# B&R Automation Studio project ABC_Pltzr
Automation Studio 3.0.90.24 SP06


## Configuration PPC70_JOB24025

CPU 4PPC70.101G-20F005, AutomationRuntime D4.22, Build 4.1.2, Vc V4.24.0, Safety 0.0

### Hardware
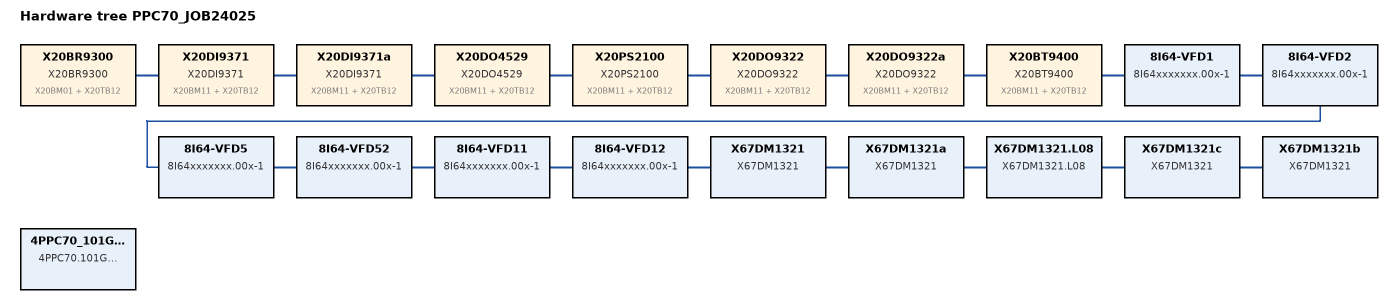
```
4PPC70_101G_20F005 : 4PPC70.101G-20F005 v1.1.0.0
  Connector IF1:
    ActivatePowerlink = 0
  Connector IF2:
    ActivateDevice = 1
    Mode = Manual
    InternetAddress = 192.168.1.100
    SubnetMask = 255.255.255.0
    InaNodeNumber = 1
    Vnc1
    VncVcObjectName1 = WSVGA
    VncKeyMappingFile1 = VC\PS2-Keyboard.dis
    VncAuthentication1 = 1
    VncPasswordViewOnly1 = v
    VncPasswordViewControl1 = 24025
    VncMaxConnections1 = 2
    VncRefreshRate1 = 500
  PermanentPvSize = 1000
  RemanentGlobalPvSize = 25000
  VolatileGlobalPvSize = 200000
  EnableUsbRemoteInstall = 1
  TimerDeviceType = SWIOTIMER
  Cyclic1Duration = 4000
  Cyclic1Tolerance = 4000
  Cyclic2Duration = 20000
  Cyclic2Tolerance = 20000
  Cyclic3Duration = 50000
  Cyclic3Tolerance = 50000
  Cyclic4Duration = 100000
  Cyclic4Tolerance = 100000
  Cyclic5Duration = 200000
  Cyclic5Tolerance = 200000
  Cyclic6Duration = 500000
  Cyclic6Tolerance = 500000
  Cyclic7Duration = 1000000
  Cyclic7Tolerance = 1000000
  Cyclic8Duration = 10000
  Cyclic8Tolerance = 30000000
  FtpUser1
  FtpUsername1 = abc
  FtpUserPassword1 = veVz20Da1KUF2Vww53L6omFNdzfk8lHY0HjcrjfOb/w=  // abc123
  FtpUserSalt1 = pyAcjG26
  FTPPath1 = 5
  FTPAccessRight1 = 0
  VcObjectName = WSVGA
  KeyMappingFile = VC\4PPC70_101G_20F005.dis
8I64-VFD1 : 8I64xxxxxxx.00x-1 v1.3.8.1  [X2X1 -> X20BT9400.X2X1]
  FunctionModel = Standard
  Supervision = off
  enableIOLR = off
  enableDigitalOutput = off
  DigitalOutputMode01 = actionDO
  ACC = 1
  DEC = 1
  HSP = 900
  ITH = 28
  BFR = 1
  UNS = 460
  FRS = 600
  NCR = 28
  NSP = 1750
  COS = 80
  TFR = 900
  DO = 9
  BRA = 0
  BLC = 64
  BRT = 15
  BEN = 0
  BET = 15
8I64-VFD11 : 8I64xxxxxxx.00x-1 v1.3.8.1  [X2X1 -> 8I64-VFD52.X2X2]
  FunctionModel = Standard
  Supervision = off
  enableIOLR = off
  enableDigitalOutput = off
  DigitalOutputMode01 = actionDO
  DownloadParameters = yes
  ACC = 1
  DEC = 1
  HSP = 900
  ITH = 13
  FTD = 600
  BFR = 1
  UNS = 460
  FRS = 600
  NCR = 13
  NSP = 1750
  COS = 80
  TFR = 900
  DO = 9
  BRA = 0
  BLC = 64
  BRT = 5
  BEN = 0
  BET = 5
8I64-VFD12 : 8I64xxxxxxx.00x-1 v1.3.8.1  [X2X1 -> 8I64-VFD11.X2X2]
  FunctionModel = Standard
  Supervision = off
  enableIOLR = off
  enableDigitalOutput = off
  DigitalOutputMode01 = actionDO
  DownloadParameters = yes
  ACC = 1
  DEC = 200
  HSP = 900
  ITH = 13
  FTD = 600
  BFR = 1
  UNS = 460
  FRS = 600
  NCR = 13
  NSP = 1750
  COS = 80
  TFR = 900
  DO = 9
  BRA = 0
  BLC = 64
  BRT = 5
  BEN = 0
  BET = 5
8I64-VFD2 : 8I64xxxxxxx.00x-1 v1.3.8.1  [X2X1 -> 8I64-VFD1.X2X2]
  FunctionModel = Standard
  Supervision = off
  enableIOLR = off
  enableDigitalOutput = off
  DigitalOutputMode01 = actionDO
  DownloadParameters = yes
  ACC = 1
  DEC = 1
  HSP = 900
  BFR = 1
  UNS = 460
  FRS = 600
  NCR = 13
  NSP = 1750
  TFR = 900
  DO = 9
  BRA = 0
  BLC = 64
  BRT = 5
  BEN = 0
  BET = 5
8I64-VFD5 : 8I64xxxxxxx.00x-1 v1.3.8.1  [X2X1 -> 8I64-VFD2.X2X2]
  FunctionModel = Standard
  Supervision = off
  DownloadParameters = yes
  ACC = 1
  DEC = 1
  HSP = 900
  ITH = 13
  FTD = 600
  BFR = 1
  UNS = 460
  FRS = 600
  NCR = 13
  NSP = 1750
  COS = 80
  TFR = 900
  DE2 = 10
  BRA = 0
8I64-VFD52 : 8I64xxxxxxx.00x-1 v1.3.8.1  [X2X1 -> 8I64-VFD5.X2X2]
  FunctionModel = Standard
  Supervision = off
  enableIOLR = off
  enableDigitalOutput = off
  DigitalOutputMode01 = actionDO
  ACC = 1
  DEC = 1
  HSP = 900
  ITH = 13
  FTD = 600
  BFR = 1
  UNS = 460
  FRS = 600
  NCR = 13
  NSP = 1750
  COS = 80
  TFR = 900
  DO = 9
  INR = 0
  BRA = 0
  BLC = 64
  BRT = 1
  BEN = 0
  BET = 1
X20BM01 : X20BM01 v1.0.0.1
X20BM11 : X20BM11 v1.0.0.0  [X2X1 -> X20BM01.X2X2]
X20BM11a : X20BM11 v1.0.0.0  [X2X1 -> X20BM11.X2X2]
X20BM11b : X20BM11 v1.0.0.0  [X2X1 -> X20BM11a.X2X2]
X20BM11c : X20BM11 v1.0.0.0  [X2X1 -> X20BM11b.X2X2]
X20BM11d : X20BM11 v1.0.0.0  [X2X1 -> X20BM11c.X2X2]
X20BM11e : X20BM11 v1.0.0.0  [X2X1 -> X20BM11f.X2X2]
X20BM11f : X20BM11 v1.0.0.0  [X2X1 -> X20BM11d.X2X2]
X20BR9300 : X20BR9300 v1.0.2.6  [SS1 -> X20TB12.SS; SL -> X20BM01.SL1; X2X1 -> 4PPC70_101G_20F005.IF5]
  Supervision = off
X20BT9400 : X20BT9400 v1.0.1.3  [SS1 -> X20TB12f.SS; SL -> X20BM11e.SL1]
  Supervision = off
X20DI9371 : X20DI9371 v1.0.1.2  [SS1 -> X20TB12a.SS; SL -> X20BM11.SL1]
  Supervision = off
X20DI9371a : X20DI9371 v1.0.1.2  [SS1 -> X20TB12b.SS; SL -> X20BM11a.SL1]
  Supervision = off
  InputFilter = 100
X20DO4529 : X20DO4529 v1.0.1.2  [SS1 -> X20TB12c.SS; SL -> X20BM11b.SL1]
  Supervision = off
X20DO9322 : X20DO9322 v1.0.2.2  [SS1 -> X20TB12e.SS; SL -> X20BM11d.SL1]
  Supervision = off
X20DO9322a : X20DO9322 v1.0.2.2  [SS1 -> X20TB12g.SS; SL -> X20BM11f.SL1]
  Supervision = off
X20PS2100 : X20PS2100 v1.0.3.0  [SS1 -> X20TB12d.SS; SL -> X20BM11c.SL1]
  Supervision = off
X20TB12 : X20TB12 v1.0.0.0
X20TB12a : X20TB12 v1.0.0.0
X20TB12b : X20TB12 v1.0.0.0
X20TB12c : X20TB12 v1.0.0.0
X20TB12d : X20TB12 v1.0.0.0
X20TB12e : X20TB12 v1.0.0.0
X20TB12f : X20TB12 v1.0.0.0
X20TB12g : X20TB12 v1.0.0.0
X67DM1321 : X67DM1321 v1.1.1.0  [X2X1 -> 8I64-VFD12.X2X2]
  Supervision = off
X67DM1321.L08 : X67DM1321.L08 v1.1.2.0  [X2X1 -> X67DM1321a.X2X2]
  Supervision = off
  Direction01 = output
  Direction02 = output
  Direction03 = output
  Direction04 = output
  Direction05 = output
  Direction06 = output
  Direction07 = output
  Direction08 = output
  Direction09 = output
  Direction10 = output
  Direction11 = output
  Direction12 = output
X67DM1321a : X67DM1321 v1.1.1.0  [X2X1 -> X67DM1321.X2X2]
  Supervision = off
  Direction01 = output
  Direction02 = output
  Direction03 = output
  Direction04 = output
X67DM1321b : X67DM1321 v1.1.1.0  [X2X1 -> X67DM1321c.X2X2]
  Supervision = off
X67DM1321c : X67DM1321 v1.1.1.0  [X2X1 -> X67DM1321.L08.X2X2]
  Supervision = off
  Direction01 = output
  Direction02 = output
```


## Logical view

Binary libraries used (declarations not repeated): astime, DataObj, Ethernet, MpCom 1.20.3, sys_lib, CSV_File

### appConfigAndRecipes.var
```iecst
(********************************************************************
 * COPYRIGHT --
 ********************************************************************
 * Package: ConfigAndRecipes
 * File: ConfigAndRecipes.var
 * Author: goran_2
 * Created: August 06, 2011
 ********************************************************************
 * Variables of package ConfigAndRecipes
 ********************************************************************)
VAR RETAIN
	gRecipe : paiRecipeApp_typ := (0);
END_VAR
VAR
	gPVSerDesMgr : paiPVSerDesMgr_typ := (0);
	gSerDesHMI_gConfigApp : paiPVSerDesHMI_typ := (0);
	gSerDesHMI_gPalletCfg : paiPVSerDesHMI_typ := (0);
	gSerDesMem_gConfigApp : configApp_typ := (0);
	gSerDesMem_gLayerEditor : palleteCfgLayer_typ := (0);
	gSerDesMem_gPallete_palCfg : palleteCfg_typ := (0);
	gDummy : UDINT := 0;
END_VAR
```

### appCfgRecDefault.h
```c
/********************************************************************
 * COPYRIGHT -- HP
 ********************************************************************
 * Program: cfgFS
 * File: cfgFSApp.h
 * Author: goran
 * Created: March 19, 2014
 *******************************************************************/

#include <bur/plctypes.h>

/*
###############################################################################
Defines, Consts
###############################################################################
*/
/*
NOTE: Using C: disk is not the best solution considering that system files are there.
However, using disk other then C: (i.e. D:, etc) for application stuff creates
issue with the ability to view/copy/access application files from windows (multiple partitions not supported, etc)

File structure used in this application is following:

Directory:
C://Data
is used for application specific stuff.
This directory holds following files:
machine configuration file - "appcfg.txt"
machine factory deafult configuration file - "appcfgfactory.txt");

a subdirectory (REC) of the above directory is used for storing recipes.
C://Data/Rec

*/

#define APP_FILE_SIZE_MAX  30000 //max file size for any recipe or config file

#define APP_DIR_NAME "Data" //root app directory; Example: C://Data
#define APP_REC_DIR_NAME "Rec" // recipes directory; Example "C://Data/Rec"

#define APP_FILENAME_CFG "appcfg.txt"
#define APP_FILENAME_CFGDEFAULT "appcfgfactory.txt"
#define APP_FILENAME_CURRECIPE "apprec.txt"
```

### Alarms.typ
```iecst
(********************************************************************

 * COPYRIGHT -- Piedmont Automation Inc.

 ********************************************************************

 * File: Alarms.typ

 * Author: goran

 * Created: Jun 1, 2015

 ********************************************************************

 * Data types for project : Alarms

 ********************************************************************)

TYPE
	applicationAlarms_enums :
		(
		APP_ALARM_HWMODULE := 0,
		APP_ALARM_DS1,
		APP_ALARM_DS2,
		APP_ALARM_DS3,
		APP_ALARM_DS4,
		APP_ALARM_DS5,
		APP_ALARM_DS6,
		APP_ALARM_ESTOP1,
		APP_ALARM_ESTOP2,
		APP_ALARM_ESTOP3,
		APP_ALARM_ESTOP4,
		APP_ALARM_ESTOP5,
		APP_ALARM_ESTOP6,
		APP_ALARM_MOTOROL,
		APP_ALARM_MCR,
		APP_ALARM_AIRPRESSURE,
		APP_ALARM_ELEV_CHAINSLACK_LF,
		APP_ALARM_ELEV_CHAINSLACK_RT,
		APP_ALARM_ELEV_PALLETDISPENS,
		APP_ALARM_VFD,
		APP_ALARM_LIGHT_CURTAIN_OSSD1,
		APP_ALARM_LIGHT_CURTAIN_OSSD2,
		APP_ALARM_INFEED_JAM,
		APP_ALARM_ROW_FORMING_JAM,
		APP_ALARM_ROW_TOO_LONG,
		APP_ALARM_INVALID_PROGRAM,
		APP_ALARM_PALLET_EXIT_TIMEOUT,
		APP_ALARM_INFEED_CASE_COUNT,
		APP_ALARM_LASTTOCHECK := 48,
		APP_ALARM_ALARMACKNEEDED := 49,
		APP_ALARM_LAST := 50
		);
END_TYPE

(*########################################################################*)
(*Application object - Alarm Object*)
(*########################################################################*)

TYPE
	applicationAlarms_typ : 	STRUCT
		oIsAlarmActiveCount : UDINT; (*1-if alarm present*)
		oIsAlarmNotAckCount : UDINT; (*1-if not ack alarm present*)
		oIsAlarmActive : BOOL; (*1-if alarm present*)
		oIsAlarmNotAck : BOOL; (*1-if not ack alarm present*)
		alarmActive : ARRAY[0..APP_ALARM_LAST]OF BOOL; (*Alarms matrix. (see Visual Components Alarm System)*)
		alarmAck : ARRAY[0..APP_ALARM_LAST]OF BOOL; (*Alarms ack matrix. (see Visual Components Alarm System)*)
	END_STRUCT;
END_TYPE
```

- appOffOnColor.clm (not shown)

- lightFeature.clm (not shown)

- pageTabs.clm (not shown)

- paiPingStatus.clm (not shown)

- Arial12px.fninfo (not shown)

- Arial7px.fninfo (not shown)

- Status_0.fninfo (not shown)

- paiHmiMenu.layer (not shown)

### sscanf2.h
```c
/********************************************************
*	NAME	: sscanf2.h
*	FUNCTION: Headerfile for the sscanf2.a implementation
*			  of the standard "C" function: sscanf().
*********************************************************/

extern int sscanf2(char *s, char *fmt, ...);
```

### Program Logical/MachineControl/blades

#### Cyclic.ld
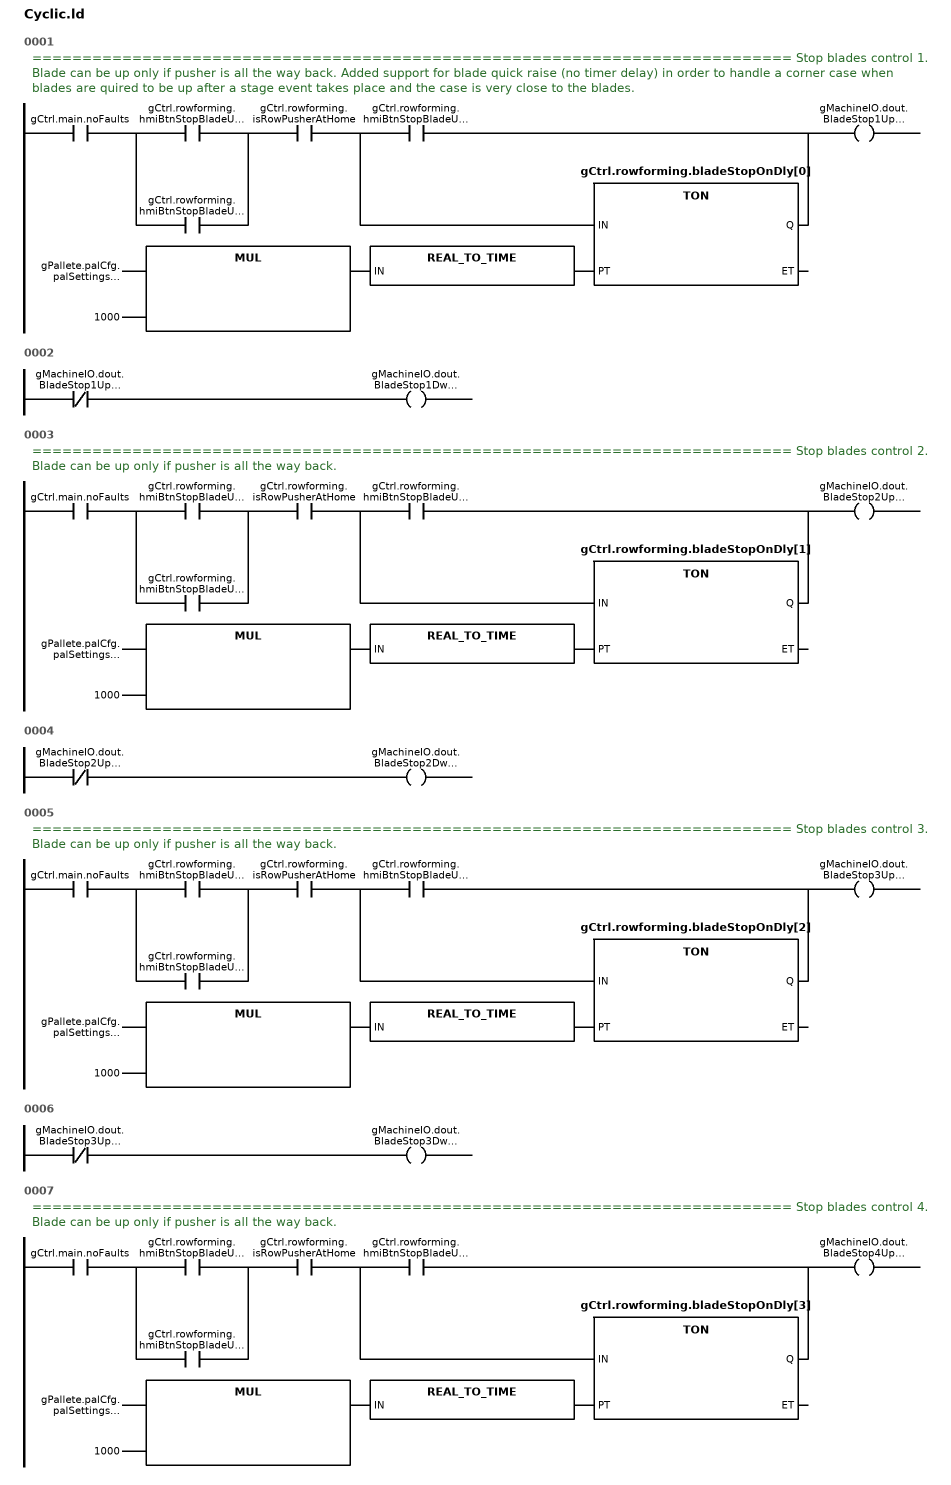
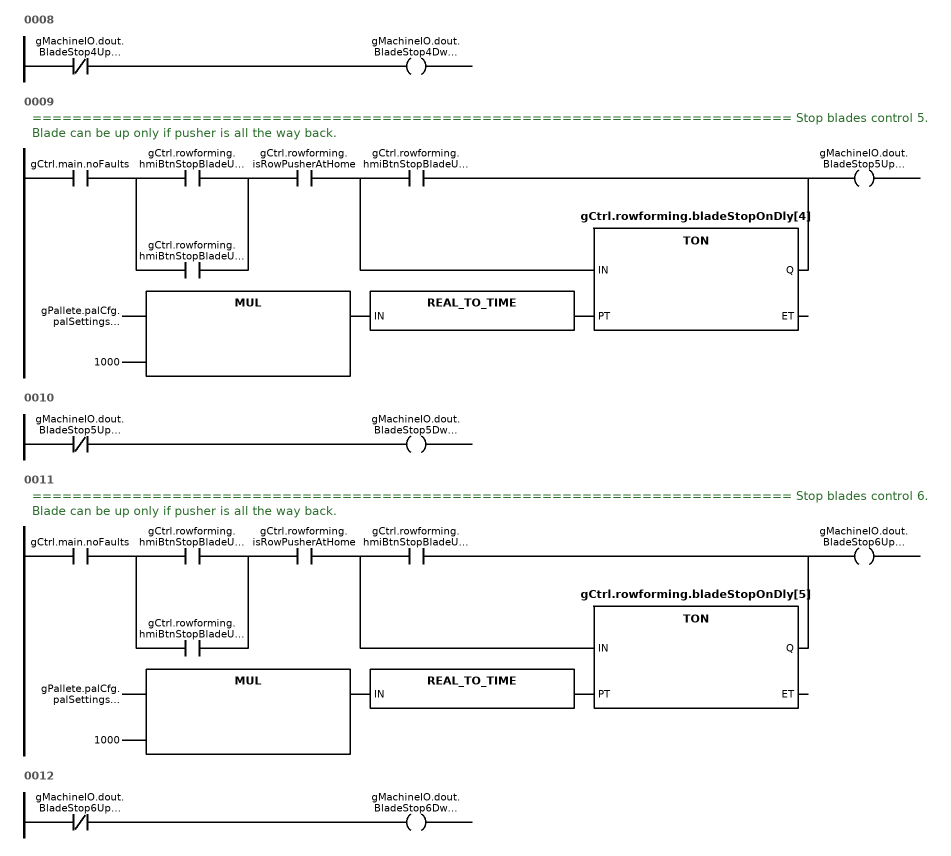
Ladder, written as Structured Text:
```iecst
PROGRAM _CYCLIC
VAR
    _p1 : BOOL;
    _p2 : BOOL;
    _p3 : BOOL;
    _p4 : BOOL;
    _p5 : BOOL;
    _p6 : BOOL;
END_VAR
(* Network 1: ============================================================================ Stop blades control 1. Blade can be up only if pusher is all the way back. Added support for blade quick raise (no timer delay) in order to handle a corner case when blades are quired to be up after a stage event takes place and the case is very close to the blades. *)
_p1 := gCtrl.main.noFaults AND (gCtrl.rowforming.hmiBtnStopBladeUpDown1 OR gCtrl.rowforming.hmiBtnStopBladeUpDownQuick1) AND gCtrl.rowforming.isRowPusherAtHome;
gMachineIO.dout.BladeStop1Up_SOL3A := (_p1 AND gCtrl.rowforming.hmiBtnStopBladeUpDownQuick1) OR gCtrl.rowforming.bladeStopOnDly[0].Q;
gCtrl.rowforming.bladeStopOnDly[0](IN := _p1, PT := REAL_TO_TIME(gPallete.palCfg.palSettings.timers.bladeStopOnDly1 * 1000));

(* Network 2 *)
gMachineIO.dout.BladeStop1Dw_SOL3B := NOT gMachineIO.dout.BladeStop1Up_SOL3A;

(* Network 3: ============================================================================ Stop blades control 2. Blade can be up only if pusher is all the way back. *)
_p2 := gCtrl.main.noFaults AND (gCtrl.rowforming.hmiBtnStopBladeUpDown2 OR gCtrl.rowforming.hmiBtnStopBladeUpDownQuick2) AND gCtrl.rowforming.isRowPusherAtHome;
gMachineIO.dout.BladeStop2Up_SOL4A := (_p2 AND gCtrl.rowforming.hmiBtnStopBladeUpDownQuick2) OR gCtrl.rowforming.bladeStopOnDly[1].Q;
gCtrl.rowforming.bladeStopOnDly[1](IN := _p2, PT := REAL_TO_TIME(gPallete.palCfg.palSettings.timers.bladeStopOnDly2 * 1000));

(* Network 4 *)
gMachineIO.dout.BladeStop2Dw_SOL4B := NOT gMachineIO.dout.BladeStop2Up_SOL4A;

(* Network 5: ============================================================================ Stop blades control 3. Blade can be up only if pusher is all the way back. *)
_p3 := gCtrl.main.noFaults AND (gCtrl.rowforming.hmiBtnStopBladeUpDown3 OR gCtrl.rowforming.hmiBtnStopBladeUpDownQuick3) AND gCtrl.rowforming.isRowPusherAtHome;
gMachineIO.dout.BladeStop3Up_SOL5A := (_p3 AND gCtrl.rowforming.hmiBtnStopBladeUpDownQuick3) OR gCtrl.rowforming.bladeStopOnDly[2].Q;
gCtrl.rowforming.bladeStopOnDly[2](IN := _p3, PT := REAL_TO_TIME(gPallete.palCfg.palSettings.timers.bladeStopOnDly3 * 1000));

(* Network 6 *)
gMachineIO.dout.BladeStop3Dw_SOL5B := NOT gMachineIO.dout.BladeStop3Up_SOL5A;

(* Network 7: ============================================================================ Stop blades control 4. Blade can be up only if pusher is all the way back. *)
_p4 := gCtrl.main.noFaults AND (gCtrl.rowforming.hmiBtnStopBladeUpDown4 OR gCtrl.rowforming.hmiBtnStopBladeUpDownQuick4) AND gCtrl.rowforming.isRowPusherAtHome;
gMachineIO.dout.BladeStop4Up_SOL6A := (_p4 AND gCtrl.rowforming.hmiBtnStopBladeUpDownQuick4) OR gCtrl.rowforming.bladeStopOnDly[3].Q;
gCtrl.rowforming.bladeStopOnDly[3](IN := _p4, PT := REAL_TO_TIME(gPallete.palCfg.palSettings.timers.bladeStopOnDly4 * 1000));

(* Network 8 *)
gMachineIO.dout.BladeStop4Dw_SOL6B := NOT gMachineIO.dout.BladeStop4Up_SOL6A;

(* Network 9: ============================================================================ Stop blades control 5. Blade can be up only if pusher is all the way back. *)
_p5 := gCtrl.main.noFaults AND (gCtrl.rowforming.hmiBtnStopBladeUpDown5 OR gCtrl.rowforming.hmiBtnStopBladeUpDownQuick5) AND gCtrl.rowforming.isRowPusherAtHome;
gMachineIO.dout.BladeStop5Up_SOL13A := (_p5 AND gCtrl.rowforming.hmiBtnStopBladeUpDownQuick5) OR gCtrl.rowforming.bladeStopOnDly[4].Q;
gCtrl.rowforming.bladeStopOnDly[4](IN := _p5, PT := REAL_TO_TIME(gPallete.palCfg.palSettings.timers.bladeStopOnDly5 * 1000));

(* Network 10 *)
gMachineIO.dout.BladeStop5Dw_SOL13B := NOT gMachineIO.dout.BladeStop5Up_SOL13A;

(* Network 11: ============================================================================ Stop blades control 6. Blade can be up only if pusher is all the way back. *)
_p6 := gCtrl.main.noFaults AND (gCtrl.rowforming.hmiBtnStopBladeUpDown6 OR gCtrl.rowforming.hmiBtnStopBladeUpDownQuick6) AND gCtrl.rowforming.isRowPusherAtHome;
gMachineIO.dout.BladeStop6Up_SOL14A := (_p6 AND gCtrl.rowforming.hmiBtnStopBladeUpDownQuick6) OR gCtrl.rowforming.bladeStopOnDly[5].Q;
gCtrl.rowforming.bladeStopOnDly[5](IN := _p6, PT := REAL_TO_TIME(gPallete.palCfg.palSettings.timers.bladeStopOnDly6 * 1000));

(* Network 12 *)
gMachineIO.dout.BladeStop6Dw_SOL14B := NOT gMachineIO.dout.BladeStop6Up_SOL14A;
END_PROGRAM
```

### Program Logical/MachineControl/elevator

#### Cyclic.ld
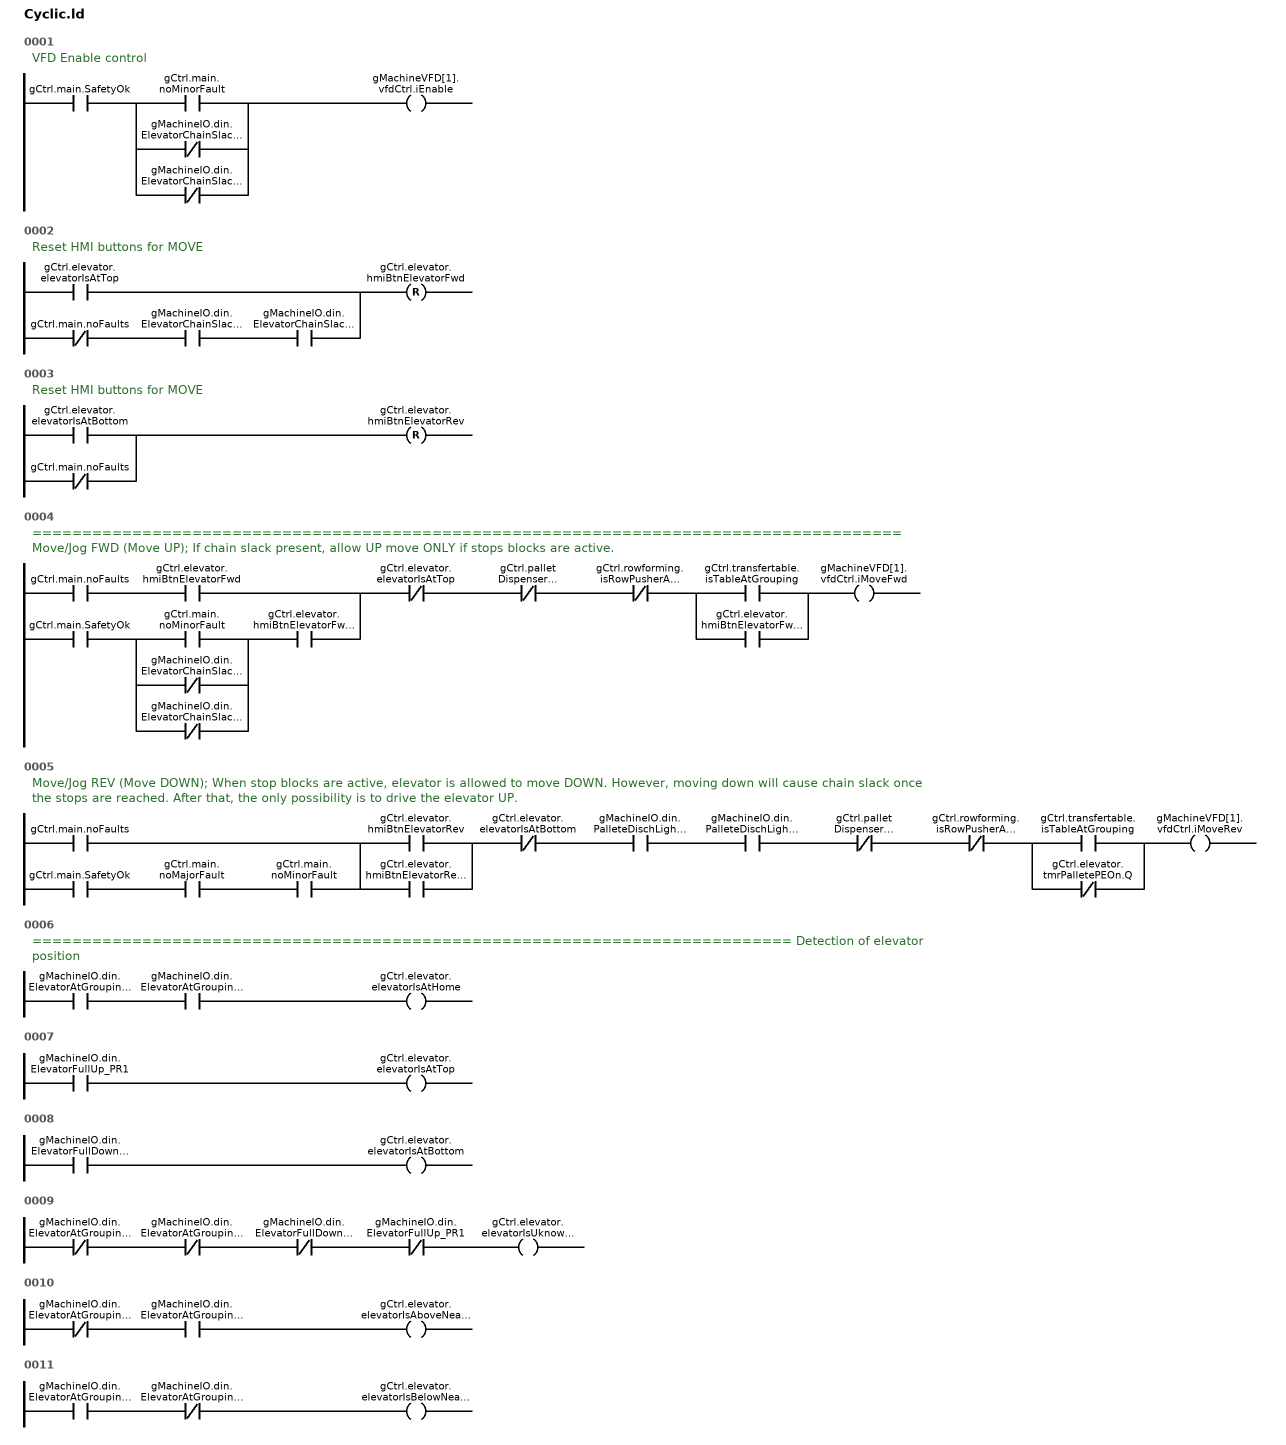
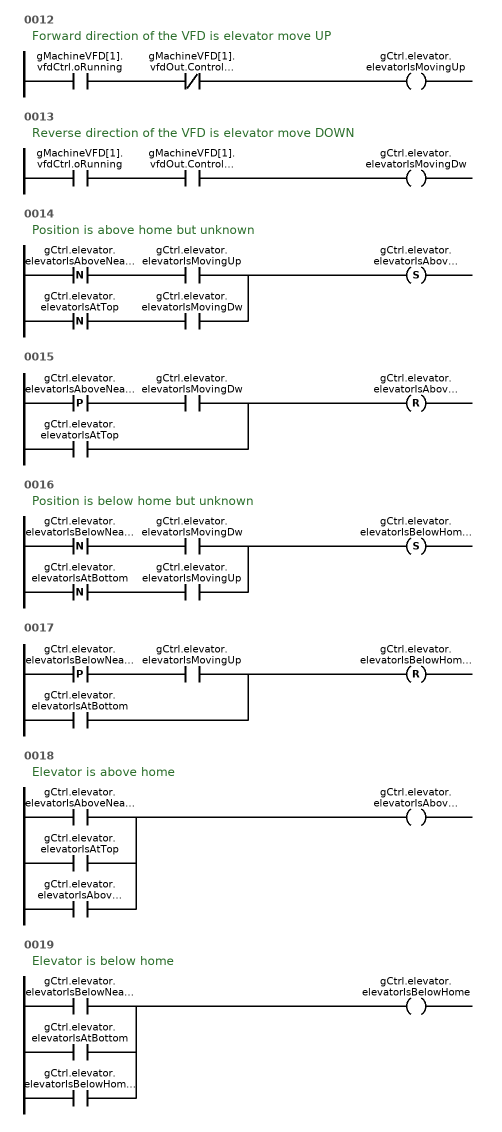
Ladder, written as Structured Text:
```iecst
PROGRAM _CYCLIC
VAR
    _p1 : BOOL;
    _p2 : BOOL;
    _p3 : BOOL;
    _e4 : F_TRIG;
    _e5 : F_TRIG;
    _e6 : R_TRIG;
    _e7 : F_TRIG;
    _e8 : F_TRIG;
    _e9 : R_TRIG;
END_VAR
(* Network 1: VFD Enable control *)
gMachineVFD[1].vfdCtrl.iEnable := gCtrl.main.SafetyOk AND (gCtrl.main.noMinorFault OR NOT gMachineIO.din.ElevatorChainSlackLF_LS7 OR NOT gMachineIO.din.ElevatorChainSlackRT_LS8);

(* Network 2: Reset HMI buttons for MOVE *)
IF gCtrl.elevator.elevatorIsAtTop OR (NOT gCtrl.main.noFaults AND gMachineIO.din.ElevatorChainSlackLF_LS7 AND gMachineIO.din.ElevatorChainSlackRT_LS8) THEN
    gCtrl.elevator.hmiBtnElevatorFwd := FALSE;
END_IF;

(* Network 3: Reset HMI buttons for MOVE *)
IF gCtrl.elevator.elevatorIsAtBottom OR NOT gCtrl.main.noFaults THEN
    gCtrl.elevator.hmiBtnElevatorRev := FALSE;
END_IF;

(* Network 4: ======================================================================================= Move/Jog FWD (Move UP); If chain slack present, allow UP move ONLY if stops blocks are active. *)
_p1 := ((gCtrl.main.noFaults AND gCtrl.elevator.hmiBtnElevatorFwd) OR (gCtrl.main.SafetyOk AND (gCtrl.main.noMinorFault OR NOT gMachineIO.din.ElevatorChainSlackLF_LS7 OR NOT gMachineIO.din.ElevatorChainSlackRT_LS8) AND gCtrl.elevator.hmiBtnElevatorFwdJog)) AND NOT gCtrl.elevator.elevatorIsAtTop AND NOT gCtrl.palletDispenser.hmiBtnPalletInCVFwd AND NOT gCtrl.rowforming.isRowPusherAtElevator;
gMachineVFD[1].vfdCtrl.iMoveFwd := _p1 AND (gCtrl.transfertable.isTableAtGrouping OR gCtrl.elevator.hmiBtnElevatorFwdJog);

(* Network 5: Move/Jog REV (Move DOWN); When stop blocks are active, elevator is allowed to move DOWN. However, moving down will cause chain slack once the stops are reached. After that, the only possibility is to drive the elevator UP. *)
_p2 := gCtrl.main.SafetyOk AND gCtrl.main.noMajorFault AND gCtrl.main.noMinorFault;
_p3 := (gCtrl.main.noFaults OR _p2) AND (gCtrl.elevator.hmiBtnElevatorRev OR gCtrl.elevator.hmiBtnElevatorRevJog) AND NOT gCtrl.elevator.elevatorIsAtBottom AND gMachineIO.din.PalleteDischLightCurtain_OSSD1 AND gMachineIO.din.PalleteDischLightCurtain_OSSD2 AND NOT gCtrl.palletDispenser.hmiBtnPalletInCVFwd AND NOT gCtrl.rowforming.isRowPusherAtElevator;
gMachineVFD[1].vfdCtrl.iMoveRev := _p3 AND (gCtrl.transfertable.isTableAtGrouping OR NOT gCtrl.elevator.tmrPalletePEOn.Q);

(* Network 6: ============================================================================ Detection of elevator position *)
gCtrl.elevator.elevatorIsAtHome := gMachineIO.din.ElevatorAtGroupingLower_PR3 AND gMachineIO.din.ElevatorAtGroupingRaise_PR4;

(* Network 7 *)
gCtrl.elevator.elevatorIsAtTop := gMachineIO.din.ElevatorFullUp_PR1;

(* Network 8 *)
gCtrl.elevator.elevatorIsAtBottom := gMachineIO.din.ElevatorFullDown_PR2;

(* Network 9 *)
gCtrl.elevator.elevatorIsUknownPosition := NOT gMachineIO.din.ElevatorAtGroupingLower_PR3 AND NOT gMachineIO.din.ElevatorAtGroupingRaise_PR4 AND NOT gMachineIO.din.ElevatorFullDown_PR2 AND NOT gMachineIO.din.ElevatorFullUp_PR1;

(* Network 10 *)
gCtrl.elevator.elevatorIsAboveNearHome := NOT gMachineIO.din.ElevatorAtGroupingLower_PR3 AND gMachineIO.din.ElevatorAtGroupingRaise_PR4;

(* Network 11 *)
gCtrl.elevator.elevatorIsBelowNearHome := gMachineIO.din.ElevatorAtGroupingLower_PR3 AND NOT gMachineIO.din.ElevatorAtGroupingRaise_PR4;

(* Network 12: Forward direction of the VFD is elevator move UP *)
gCtrl.elevator.elevatorIsMovingUp := gMachineVFD[1].vfdCtrl.oRunning AND NOT gMachineVFD[1].vfdOut.Control.Direction;

(* Network 13: Reverse direction of the VFD is elevator move DOWN *)
gCtrl.elevator.elevatorIsMovingDw := gMachineVFD[1].vfdCtrl.oRunning AND gMachineVFD[1].vfdOut.Control.Direction;

(* Network 14: Position is above home but unknown *)
_e4(CLK := gCtrl.elevator.elevatorIsAboveNearHome);
_e5(CLK := gCtrl.elevator.elevatorIsAtTop);
IF (_e4.Q AND gCtrl.elevator.elevatorIsMovingUp) OR (_e5.Q AND gCtrl.elevator.elevatorIsMovingDw) THEN
    gCtrl.elevator.elevatorIsAboveHomeUnknown := TRUE;
END_IF;

(* Network 15 *)
_e6(CLK := gCtrl.elevator.elevatorIsAboveNearHome);
IF (_e6.Q AND gCtrl.elevator.elevatorIsMovingDw) OR gCtrl.elevator.elevatorIsAtTop THEN
    gCtrl.elevator.elevatorIsAboveHomeUnknown := FALSE;
END_IF;

(* Network 16: Position is below home but unknown *)
_e7(CLK := gCtrl.elevator.elevatorIsBelowNearHome);
_e8(CLK := gCtrl.elevator.elevatorIsAtBottom);
IF (_e7.Q AND gCtrl.elevator.elevatorIsMovingDw) OR (_e8.Q AND gCtrl.elevator.elevatorIsMovingUp) THEN
    gCtrl.elevator.elevatorIsBelowHomeUnknown := TRUE;
END_IF;

(* Network 17 *)
_e9(CLK := gCtrl.elevator.elevatorIsBelowNearHome);
IF (_e9.Q AND gCtrl.elevator.elevatorIsMovingUp) OR gCtrl.elevator.elevatorIsAtBottom THEN
    gCtrl.elevator.elevatorIsBelowHomeUnknown := FALSE;
END_IF;

(* Network 18: Elevator is above home *)
gCtrl.elevator.elevatorIsAboveHome := gCtrl.elevator.elevatorIsAboveNearHome OR gCtrl.elevator.elevatorIsAtTop OR gCtrl.elevator.elevatorIsAboveHomeUnknown;

(* Network 19: Elevator is below home *)
gCtrl.elevator.elevatorIsBelowHome := gCtrl.elevator.elevatorIsBelowNearHome OR gCtrl.elevator.elevatorIsAtBottom OR gCtrl.elevator.elevatorIsBelowHomeUnknown;
END_PROGRAM
```

### Program Logical/MachineControl/vfdControl

#### vfdControl.c
```c
#include <bur/plctypes.h>

#ifdef _DEFAULT_INCLUDES
	#include <AsDefault.h>
#endif

/*
16#0000	nOF: No fault code saved
16#1000	CrF: Capacitor pre-charge detected fault or
16#1000	OLF: Motor overload or
16#1000	SOF: Motor overspeed
16#2310	OCF: Overcurrent
16#2320	OCF: Impeding short-circuit or
16#2320	OCF: Power module, specific to 15kW drives
16#2330	SCF: Motor short-circuit (to ground)
16#2340	OCF: Motor short-circuit (phase to phase)
16#3110	OSF: Line supply overvoltage
16#3120	USF: Line supply undervoltage
16#3130	PHF: Line supply phase loss
16#3310	ObF: DC bus overvoltage or
16#3310	OPF: Motor phase loss or
16#3310	OPF: Motor phase loss - 3 phases
16#4210	OHF: Drive overheating
16#5520	EEF: EEPROM memory
16#6100	InF: Internal
16#6300	CFF: Incorrect configuration (parameters) or
16#6300	CFI: Invalid configuration (parameters)
16#7300	LFF: 4 - 20 mA loss
16#7510	SLF: Modbus communication interruption
16#8100	COF: Communication interruption, line 2 (CANopen)
16#9000	EPF: External fault
16#FF00	tnF: Auto-tuning was unsuccessful
16#FF01	bLF: Brake control
16#7520	ILF: Optional internal link
16#7510	CNF: Communication interruption on the communication card
*/
static void paiVFDGetFaultText(UINT faultCode, char* pDest, UDINT destSize)
{

	switch(faultCode){
		case 0x0:
			brsstrcpy((UDINT)pDest, (UDINT)"nOF: No fault code saved");
			break;
		case 0x1000:
			brsstrcpy((UDINT)pDest, (UDINT)"CrF or OLF or SOF");
			break;
		case 0x2310:
			brsstrcpy((UDINT)pDest, (UDINT)"OCF: Overcurrent");
			break;
		case 0x2320:
			brsstrcpy((UDINT)pDest, (UDINT)"OCF: Impeding short-circuit");
			break;
		case 0x2330:
			brsstrcpy((UDINT)pDest, (UDINT)"SCF: Motor short-circuit (to ground)");
			break;
		case 0x2340:
			brsstrcpy((UDINT)pDest, (UDINT)"OCF: Motor short-circuit (phase to phase)");
			break;
		case 0x3110:
			brsstrcpy((UDINT)pDest, (UDINT)"OSF: Line supply overvoltage");
			break;
		case 0x3120:
			brsstrcpy((UDINT)pDest, (UDINT)"USF: Line supply undervoltage");
			break;
		case 0x3130:
			brsstrcpy((UDINT)pDest, (UDINT)"PHF: Line supply phase loss");
			break;
		case 0x3310:
			brsstrcpy((UDINT)pDest, (UDINT)"ObF: DC bus overvoltage or OPF");
			break;
		case 0x4210:
			brsstrcpy((UDINT)pDest, (UDINT)"OHF: Drive overheating");
			break;
		case 0x5520:
			brsstrcpy((UDINT)pDest, (UDINT)"EEF: EEPROM memory");
			break;
		case 0x6100:
			brsstrcpy((UDINT)pDest, (UDINT)"InF: Internal");
			break;
		case 0x6300:
			brsstrcpy((UDINT)pDest, (UDINT)"CFF: Incorrect configuration or CFI");
			break;
		case 0x7300:
			brsstrcpy((UDINT)pDest, (UDINT)"LFF: 4 - 20 mA loss");
			break;
		case 0x7510:
			brsstrcpy((UDINT)pDest, (UDINT)"SLF: Modbus communication interruption");
			break;
		case 0x8100:
			brsstrcpy((UDINT)pDest, (UDINT)"COF: Communication interruption, line 2 (CANopen)");
			break;
		case 0x9000:
			brsstrcpy((UDINT)pDest, (UDINT)"EPF: External fault");
			break;
		case 0xFF00:
			brsstrcpy((UDINT)pDest, (UDINT)"tnF: Auto-tuning was unsuccessful");
			break;
		case 0xFF01:
			brsstrcpy((UDINT)pDest, (UDINT)"bLF: Brake control");
			break;
		default:
			brsstrcpy((UDINT)pDest, (UDINT)"Unknown fault");
			break;
	}
}

static void paiVFDShutOff(paiVFD_typ* p)
{
	p->vfdOut.Control.DisableVoltage = 0;
	p->vfdOut.Control.SwitchOn = 0;
	p->vfdOut.Control.VelocitySetpoint = 0;
	p->vfdOut.Control.EnableOperation = 0;
	p->vfdOut.Control.QuickStop = 0;

	p->vfdCtrl.oFault = 0;
	p->vfdCtrl.oReady = 0;
	p->vfdCtrl.oRunning = 0;

	if(!p->vfdIn.ModuleInfo.ModuleOk){
		brsstrcpy((UDINT)p->stateText, (UDINT)"Not present");
	}else{
		brsstrcpy((UDINT)p->stateText, (UDINT)"Off Line");
	}
}

static void paiVFDCyclic(paiVFD_typ* p)
{
	if(!p)
		return;

	if(!p->vfdIn.ModuleInfo.ModuleOk || !p->vfdCtrl.iVoltageEnable){
		paiVFDShutOff(p);
		return;
	}

//	if(!p->vfdCtrl.iEnable){
//		paiVFDShutOff(p);
//		return;
//	}

	p->vfdOut.Control.DisableVoltage = 1;
	p->vfdOut.Control.QuickStop = !p->vfdCtrl.iEStop;
	p->vfdOut.Control.SwitchOn = p->vfdIn.Status.ReadyToSwitchOn;
//	p->vfdOut.Control.EnableOperation = p->vfdIn.Status.SwitchedOn & ( (p->vfdCtrl.iEnable & p->vfdCtrl.iMoveFwd) || ((p->vfdCtrl.iEnable & p->vfdCtrl.iMoveRev)) );

	//IMPORTANT: work around for getting the drive to stop very quickly. No decel would stop it!
#if 0
	if(p->appID == 6){
		p->vfdOut.Control.EnableOperation = p->vfdIn.Status.SwitchedOn & p->vfdCtrl.iEnable & (p->vfdCtrl.iMoveFwd || p->vfdCtrl.iMoveRev /*|| (p->vfdIn.Status.CurrentVelocity != 0)*/ );
	}else{
		p->vfdOut.Control.EnableOperation = p->vfdIn.Status.SwitchedOn & p->vfdCtrl.iEnable & (p->vfdCtrl.iMoveFwd || p->vfdCtrl.iMoveRev || (p->vfdIn.Status.CurrentVelocity != 0) );
	}
#endif
	//Following code allows stopping very fast if dec set to 1. Otherwise, the VFD decel ramp is used; Only used for VFD2 and VFD52
	if(  ((p->appID == 6) /*&& (gPaiVFDX64Mgr.mX64VFDs[3].mX64Params[1].oValue == 1)*/) || //VFD52
		 ((p->appID == 2) && (gPaiVFDX64Mgr.mX64VFDs[1].mX64Params[1].oValue == 1)) || //VFD2
		 ((p->appID == 5) && (gPaiVFDX64Mgr.mX64VFDs[2].mX64Params[1].oValue == 1))  //VFD5
		){
		p->vfdOut.Control.EnableOperation = p->vfdIn.Status.SwitchedOn & p->vfdCtrl.iEnable & (p->vfdCtrl.iMoveFwd || p->vfdCtrl.iMoveRev /*|| (p->vfdIn.Status.CurrentVelocity != 0)*/ );
	}else{
		p->vfdOut.Control.EnableOperation = p->vfdIn.Status.SwitchedOn & p->vfdCtrl.iEnable & (p->vfdCtrl.iMoveFwd || p->vfdCtrl.iMoveRev || (p->vfdIn.Status.CurrentVelocity != 0) );
	}

	//p->vfdOut.Control.EnableOperation = p->vfdIn.Status.SwitchedOn & p->vfdCtrl.iEnable;
	//	p->vfdOut.Control.RunAsked = p->vfdCtrl.iMoveFwd || p->vfdCtrl.iMoveRev;
	if(p->vfdCtrl.iMoveFwd){
		p->vfdOut.Control.Direction = 0;
	}else
	if(p->vfdCtrl.iMoveRev){
		p->vfdOut.Control.Direction = 1;
	}else{
		p->vfdOut.Control.Direction = 0;
	}

	if(p->vfdCtrl.iMoveRev || p->vfdCtrl.iMoveFwd){
		p->vfdOut.Control.VelocitySetpoint = p->vfdCtrl.iVelocitySetPoint;
	}else{
		p->vfdOut.Control.VelocitySetpoint = 0;
	}

	//p->vfdOut.Control.VelocitySetpoint = p->vfdCtrl.iVelocitySetPoint;
	p->vfdOut.Control.FaultReset = p->vfdCtrl.iFaultReset;
	p->vfdCtrl.oFault = p->vfdIn.Status.FaultDetection;
	p->vfdCtrl.oReady = p->vfdIn.Status.SwitchedOn;
	p->vfdCtrl.oRunning = (p->vfdIn.Status.CurrentVelocity != 0) ? 1 : 0;

	if(!p->vfdIn.Status.SwitchedOn){
		brsstrcpy((UDINT)p->stateText, (UDINT)"Not ready");
	}else
	if(p->vfdIn.Status.FaultDetection){
		brsstrcpy((UDINT)p->stateText, (UDINT)"Fault");
		paiVFDGetFaultText(p->vfdIn.Fault.CurrentFault, &p->vfdIn.Fault.CurrentFaultTxt[0], 63);
	}else
	if(p->vfdCtrl.oRunning){
		char velocityRpmTxt[32];
		brsitoa((UDINT)p->vfdIn.Status.CurrentVelocity, (UDINT)velocityRpmTxt);
		if(p->vfdIn.Status.CurrentVelocity > 0){
			brsstrcpy((UDINT)p->stateText, (UDINT)"MoveFwd @ ");
			brsstrcat((UDINT)p->stateText, (UDINT)velocityRpmTxt);
			brsstrcat((UDINT)p->stateText, (UDINT)"[rpm]");
		}else{
			brsstrcpy((UDINT)p->stateText, (UDINT)"MoveRev @ ");
			brsstrcat((UDINT)p->stateText, (UDINT)velocityRpmTxt);
			brsstrcat((UDINT)p->stateText, (UDINT)"[rpm]");
		}
	}else{
		brsstrcpy((UDINT)p->stateText, (UDINT)"Stopped");
	}
}

/*
###############################################################################
Init, Cyclic, Exit
###############################################################################
*/
void _INIT vfdControlInit(void)
{
	int ii;

	//on power up > remove all VFD-s, make them "not present"
	for(ii=0; ii<=APP_VFD_IDXLAST;ii++){
		gMachineVFD[ii].vfdCtrl.iVoltageEnable = 0;
		brsstrcpy((UDINT)gMachineVFD[ii].description, (UDINT)"unused VFD control entry");
	}

	//define, designate and allow operation for VFD-s that are used in this application

	//IMPORTANT: VFD1 is configured to automaticaly control VFD DO (digital output) as a break control output
	//see VFD configuration; param BLC is set to DO
//	gMachineVFD[1].vfdCtrl.iVoltageEnable = 1;
	brsstrcpy((UDINT)gMachineVFD[1].description, (UDINT)"VFD1-Elevator");

	//IMPORTANT: VFD2 is configured to automaticaly control VFD DO (digital output) as a break control output
	//see VFD configuration; param BLC is set to DO
//	gMachineVFD[2].vfdCtrl.iVoltageEnable = 1;
	brsstrcpy((UDINT)gMachineVFD[2].description, (UDINT)"VFD2-Transfer Table");

	//IMPORTANT: VFD4 is configured to automaticaly control VFD DO (digital output) as a break control output
	//see VFD configuration; param BLC is set to DO
//	gMachineVFD[4].vfdCtrl.iVoltageEnable = 1;
//	brsstrcpy((UDINT)gMachineVFD[4].description, (UDINT)"VFD4-Row Pusher");
	brsstrcpy((UDINT)gMachineVFD[5].description, (UDINT)"VFD5-RowFormingRollers");
	brsstrcpy((UDINT)gMachineVFD[6].description, (UDINT)"VFD52-RowFormingRollers");

//	gMachineVFD[11].vfdCtrl.iVoltageEnable = 1;
	brsstrcpy((UDINT)gMachineVFD[11].description, (UDINT)"VFD11-Palletizing Mesh CV");
	brsstrcpy((UDINT)gMachineVFD[12].description, (UDINT)"VFD11-Discharge Mesh CV");
}

void _CYCLIC vfdControlCyclic(void)
{
	int ii;

	//cyclicly copy VFD HW status to the VFD control structure
	//Note:
	//VFD1 (designated in the schematic under that name) has an X2X address 8 (station 8). See X2X network diagram
	//VFD2 (designated in the schematic under that name) has an X2X address 9 (station 9). See X2X network diagram
	//etc
	brsmemcpy((UDINT)&gMachineVFD[1].vfdIn.ModuleInfo, (UDINT)&gHWModules[9], sizeof(gMachineVFD[1].vfdIn.ModuleInfo));
	brsmemcpy((UDINT)&gMachineVFD[2].vfdIn.ModuleInfo, (UDINT)&gHWModules[10], sizeof(gMachineVFD[1].vfdIn.ModuleInfo));
	//brsmemcpy((UDINT)&gMachineVFD[4].vfdIn.ModuleInfo, (UDINT)&gHWModules[11], sizeof(gMachineVFD[1].vfdIn.ModuleInfo));
	brsmemcpy((UDINT)&gMachineVFD[5].vfdIn.ModuleInfo, (UDINT)&gHWModules[11], sizeof(gMachineVFD[1].vfdIn.ModuleInfo));
	brsmemcpy((UDINT)&gMachineVFD[6].vfdIn.ModuleInfo, (UDINT)&gHWModules[12], sizeof(gMachineVFD[1].vfdIn.ModuleInfo));
	brsmemcpy((UDINT)&gMachineVFD[11].vfdIn.ModuleInfo, (UDINT)&gHWModules[13], sizeof(gMachineVFD[1].vfdIn.ModuleInfo));
	brsmemcpy((UDINT)&gMachineVFD[12].vfdIn.ModuleInfo, (UDINT)&gHWModules[14], sizeof(gMachineVFD[1].vfdIn.ModuleInfo));

	gMachineVFD[1].vfdCtrl.iVoltageEnable = gCtrl.main.EStopOk;
	gMachineVFD[2].vfdCtrl.iVoltageEnable = gCtrl.main.EStopOk;
	//gMachineVFD[4].vfdCtrl.iVoltageEnable = gCtrl.main.EStopOk;
	gMachineVFD[5].vfdCtrl.iVoltageEnable = gCtrl.main.EStopOk;
	gMachineVFD[6].vfdCtrl.iVoltageEnable = gCtrl.main.EStopOk;
	gMachineVFD[11].vfdCtrl.iVoltageEnable = gCtrl.main.EStopOk;
	gMachineVFD[12].vfdCtrl.iVoltageEnable = gCtrl.main.EStopOk;

	//operate IO for all VFD-s
	for(ii=0; ii<=APP_VFD_IDXLAST;ii++){
		paiVFDCyclic(&gMachineVFD[ii]);
	}
}
```

### Package Logical/paiComponents/Libraries - pai Custom static libraries

### Program Logical/paiComponents/Libraries/bgringbuf

#### bgringbuffer.c
```c
#ifndef _BG_RINGBUFFER_C
#define _BG_RINGBUFFER_C
/*
File:
bgRingBuffer.c

About:
------
- ring buffer implementation

B&R System Dependencies:
------------------------
- B&R system library: none
- B&R system header files: stdarg.h

History:
--------
06/26/2015
-created static c/c++ library version

03/11/2005
-first version

Test and example code:
----------------------
- to run this file standalone:
--- enable following code section (remove or comment out #if 0 / #endif)
--- create cyclic object (task) from C Language and add this file
*/
#include <stdarg.h>

#include <bur/plctypes.h>
#ifdef _DEFAULT_INCLUDES
	#include <AsDefault.h>
#endif

#include "bgringbuffer.h"
#include "../sprintf2/sprintf2.h"

#if 0
#include<bur/plc.h>
#include <bur/plctypes.h>

//#include <bgsprintf.h>
#include <bgringbuffer.h>

_LOCAL int counter;

_LOCAL bgRingBuffer_typ myRB;

#define TXT_SIZE 64
_LOCAL char textBuffer1[TXT_SIZE];
_LOCAL char textBuffer2[TXT_SIZE];

#define RB_SIZE 64
_LOCAL char ringBuffer[RB_SIZE];

_INIT void Init(void) {

	rbInit(&myRB, ringBuffer, RB_SIZE);
}

_CYCLIC void Cyclic(void) {

	counter++;

	sprintf2(textBuffer1, "Counter=%d\n", counter);
	bgRingBuffPutString(&myRB, textBuffer1);
    bgRingBuffGet(&myRB, textBuffer2, TXT_SIZE);
}
#endif
/*End: Example/Test code*/

static char *bgRingBuffGetPtrToFileName(char *pFileNameWithPath)
{
/*
Input Example:
*pFileNameWithPath = "d:/data/temp/cobble/2005-9-1/new_ng.pgp/pgm/new_ng/cpu/bgstatemachine.c"
                                                                             |
Output value is ptr to: bgstatemachine.c ------------------------------------+
*/
int i;
int len = brsstrlen((UDINT)pFileNameWithPath);
char* pStart = (char*)(pFileNameWithPath + len);
	for(i=0;i<len; i++, pStart--){
		if( (*pStart == '/') || (*pStart == '\\') ){
			pStart++;
			return pStart;
		}
	}
	return pFileNameWithPath;
}

static void bgRingBuffIncDataInPtr(bgRingBuffer_typ *rb){
	rb->ptrDataIn++;
    if(rb->ptrDataIn >= rb->ptrCircularBufferEnd){
    	rb->ptrDataIn = rb->ptrCircularBufferBegin;
#if 0
/*mark wrap arround for testing*/
    	*rb->ptrDataIn = '@';
    	rb->ptrDataIn++;
#endif
    }
}

static void bgRingBuffIncDataOutPtr(bgRingBuffer_typ *rb){
	rb->ptrDataOut++;
	if(rb->ptrDataOut >= rb->ptrCircularBufferEnd)
		rb->ptrDataOut = rb->ptrCircularBufferBegin;
}

void bgRingBuffInit(bgRingBuffer_typ *rb, char *buffer, int bufSize)
{
	if(!buffer || !bufSize)
		return;

	rb->init = 1;
	rb->overrun = 0;
	rb->bufSize = bufSize;
    rb->ptrCircularBufferBegin = buffer;
    rb->ptrCircularBufferEnd = buffer + rb->bufSize;
    rb->ptrDataIn = rb->ptrCircularBufferBegin;
    rb->ptrDataOut = rb->ptrCircularBufferBegin;
}
/*
----------------------------------------------------------
*/
void bgRingBuffPutString(bgRingBuffer_typ *rb, char *sourceString)
{
    char *src = sourceString;

	if(!rb->init)
		return;

    /*input is string! look for zero termination*/
    while( *src ){

        /*store char*/
        *rb->ptrDataIn = *src;

        /*inc ptrs*/
		src++;

        bgRingBuffIncDataInPtr(rb);

        /*check if ring-buffer full*/
        if(rb->ptrDataIn == rb->ptrDataOut){
        	/*move out ptr one step ahead of in ptr*/
	        bgRingBuffIncDataOutPtr(rb);

			/*mark ring buffer overrun*/
			if(!rb->overrun){
		        char text[3]={'<','?','>'};
		        int i;
				rb->overrun = 1;
	        	for(i=0;i<3;i++){
			        *rb->ptrDataIn = text[i];
			        bgRingBuffIncDataInPtr(rb);
			        bgRingBuffIncDataOutPtr(rb);
		        }
		    }
        }
    }
}
/*
----------------------------------------------------------
*/
int bgRingBuffGet(bgRingBuffer_typ *rb, char *destination, int destSize)
{
char *dst = destination;
char *dstMax = dst + destSize;
int length = 0;

	if(!rb->init)
		return 0;

    if(rb->ptrDataIn == rb->ptrDataOut)
        return 0;

    while(1){
        *dst = *rb->ptrDataOut;
		length++;

        dst++;
        /*check if max size riched*/
        if(dst >= dstMax)
            break;

  		bgRingBuffIncDataOutPtr(rb);

        /*check if ring-buffer empty*/
        if(rb->ptrDataIn == rb->ptrDataOut){

        	/*mark end of ring buffer overrun*/
			if(rb->overrun){
		        char text[3]={'<','!','>'};
		        int i;

				rb->overrun = 0;
	        	for(i=0;i<3;i++){
			        *dst = text[i];
			        dst++;
			        length++;
			        if(dst >= dstMax)
			            break;
		        }
		    }

            break;
        }
    }
    return length;
}

void bgRingBuffPutDbgInfo(bgRingBuffer_typ *rb, char *file, char *function, unsigned int level, unsigned int unused, char *format, ...)
{
char txt[512];

va_list args;

	/*if dbg entry level > then currently set dbg level -> exit*/
	if( level > rb->dbgLevel )
		return;

	/*timestap needed? default=no*/
	if( rb->dbgFormat & BG_DEBUG_FORMAT_LEVEL){
		switch(level){
			case 0: bgRingBuffPutString(rb, "CRT|"); break;
			case 1: bgRingBuffPutString(rb, "ERR|"); break;
			case 2: bgRingBuffPutString(rb, "WAR|"); break;
			case 3: bgRingBuffPutString(rb, "INF|"); break;
			case 4: bgRingBuffPutString(rb, "DBG|"); break;
			default: bgRingBuffPutString(rb, "???|"); break;
		}
	}

	/*timestap needed? default=no*/
	if( rb->dbgFormat & BG_DEBUG_FORMAT_TIMESTAMP){
		snprintf2(txt, 512, "%s|", "2005-10-01 12:32:44.123" );
		bgRingBuffPutString(rb, txt);
	}

	/*filename needed? default=no*/
	if( rb->dbgFormat & BG_DEBUG_FORMAT_FILENAME){
		snprintf2(txt, 512, "%s|", bgRingBuffGetPtrToFileName(file) );
		bgRingBuffPutString(rb, txt);
	}

	/*function name needed? default=no*/
	if( rb->dbgFormat & BG_DEBUG_FORMAT_FUNCTION){
		snprintf2(txt, 512, "%s()|", function);
		bgRingBuffPutString(rb, txt);
	}

    va_start( args, format );

	snvprintf2(txt, 512, format, args);
	//snvprintf2(txt, 512, format, args);

	va_end(args);

	bgRingBuffPutString(rb, txt);
}

void bgRingBuffPrintf(bgRingBuffer_typ *rb, char *format, ...)
{
char txt[512];
va_list ap;

    va_start( ap, format );

	snvprintf2(txt, 512, format, ap);

	va_end(ap);

	bgRingBuffPutString(rb, txt);
}

#endif
/*EOF*/
```

### Package Logical/paiComponents/bglib - pai C utilities

### bgstring.h
```c
/**\file: bgString.h
*Useful string manipulation functions.
*/
#ifndef _BG_STRING_H
#define _BG_STRING_H

#ifndef WIN32
/*B&R string functions*/
//#include <string.h>
#include <asbrstr.h>
#endif

/**
Find if string (*sub) is present within the string (*s).
Start search at (start) index, don't search beyond (end) index of input string (*s)
\param s prt to source string
\param sub prt to sub string
\param start location (s[start]) to start the search (-1:use default(start at 0) | 0..strlen(s)-1 )
\param end end search at location s[end] (-1=use default(EndOfString) OR 0..strlen(s)-1 )
\return -1 substring not found
\return >=0 index of (s) where the (sub) starts
*/
int bgStrFind(char *s, char *sub, int start, int end);

/**
Similar to bgStrFind, except for and extra option.
\param option (0-same as bgStrFind; 1-use case insensitive string compare)
\return -1 substring not found
\return >=0 index of (s) where the (sub) starts
*/
int bgStrFindEx(char *s, char *sub, int start, int end, int option);

/**
Copy up to (maxNoOfCharsToCopy) chars from (*src) string to (*dest) string.
If (*src) string is shorter then (maxNoOfCharsToCopy-1) return value will be
equal to the length of the src string.
*\return Number of bytes actually copied
*/
int bgStrCpyN(char *dest, char *src, int maxNoOfCharsToCopy);

/**
Copy up to (maxNoOfCharsToCopy) chars from (*src) string to (*dest) string and trim leading spaces when coping
If (*src) string is shorter then (maxNoOfCharsToCopy-1) return value will be
equal to the length of the src string.
*\return Number of bytes actually copied
*/
int bgStrCpyNTrimLeadingSpaces(char *dest, char *src, int maxNoOfCharsToCopy);

/**
Terminate (by writing 0) supplied string at CR or LF which ever is found first.
If oldStrLen (before calling this func) equals to the return value of this
function it means that string termination (removal of LF or CR) didn't take
place.
\return New string length
*/
int bgStrTrimCRLF(char *dest);

/**
Check if input char (c) is a digit ('0','1', to '9')
\return 0 - no
\return 1 - yes
*/
int bgIsDigit(char c);

/**
Check if input string (s) is a unsigned integer number.
Or, in other words, if all chars in the input string are digits.
\return 0 - no
\return 1 - yes
*/
int bgIsNumber_uint(char *s);

/**
Check if string is a integer (+/-) number (i.e all chars in strings are digits)
\return 0 - no
\return 1 - yes
*/
int bgIsNumber_int(char *s);

/**
Convert input string (s) to unsigned int (dst)
\return 0 - failed (input not a valid string, *dst not changed)
\return 1 - ok (*dst set to new value)
*/
int bgAsciiToUint(char *src, unsigned int *dst);

/**
Convert input string to int value
\return 0 - failed (input not a valid string, *dst not changed)
\return 1 - ok (*dst set to new value)
*/
int bgAsciiToInt(char *src, unsigned int *dst);

/**
\def BG_STRINGLIST_MAXITEMCOUNT
Defines maximum number of items (pointers) within the list of strings
*/
#define BG_STRINGLIST_MAXITEMCOUNT	512

/**
\struct bgStringList_typ
Data object that holds list of strings.\n
Typical usage is following: input/source stream (*src), that contains lines
separated by CRLF or LF, is scanned and all line ends are terminated with 0.
Pointers to the start of each line are entered into the (items) array of ptrs.\n
<b>NOTE:</b> All ptrs in (items[]) point into the space within the (*src) buffer!\n
<b>IMPORTANT:</b> Generating list of line ptrs is a destructive process as the
(*src) buffer gets modified (0 are writen at the place of each LF or CR).
*/
typedef struct bgStringList_typ
{
/*in*/
	unsigned char	*src;			/**<Input: ptr to the source stream/input buffer */
/*out*/
	int				itemCount;		/**<Output: number of items in the list*/
	unsigned char 	*items[BG_STRINGLIST_MAXITEMCOUNT]; /**<Output: list of pointers to strings*/
}bgStringList_typ;

/**
\struct bgStringListEx_typ
Data object that holds list of strings. In this case, list of ptrs (items) is supplied externally (allocate memory)\n
Typical usage: same as \link bgStringList_typ \endlink\n
<b>IMPORTANT:</b> Before using this data object, the list of items (items) must be initialized
(i.e. allocated or external memory must be assigned to (items) ptr!)\n
Use method \link bgStringListExMemSet \endlink to set the ptrs array memory.
*/
typedef struct bgStringListEx_typ
{
/*in*/
	unsigned char	*src;		/**<Input: ptr to the source stream/input buffer */
	int				itemCountMax;	/**<Input: Maximum number of items (depends on the size of externaly supplied memory*/
/*out*/
	int				itemCount;	/**<Output: number of items in the list*/
	unsigned char 	**items;	/**<Output: list of pointers to strings (memory is user supplied*/
}bgStringListEx_typ;

/**
Method for data object \link bgStringList_typ \endlink\n
\param p Ptr to data object: (\link bgStringList_typ \endlink)
Example: Given user supplied input stream (*src), i.e.:
\code
"hello world\r\nwhat is new?\r\nthird line\r\nline #4\r\n"\n
\endcode
Method generates following: (p-> points to \link bgStringList_typ \endlink data object):
\code
p->itemCount = 4; <*src> string has 4 lines
p->items[0] = ptr to 1st line ("hello world");
p->items[1] = ptr to 2nd line ("what is new?");
p->items[2] = ptr to 3rd line ("third line");
p->items[3] = ptr to 4th line ("line #4");
\endcode
\n
Method is used when processing ascii based client/server protocols (i.e. FTP, Telnet...)\n
<b>IMPORTANT:</b>Method write 0-s (string termination) into the source stream (*src) at the position of
each line end!\n
(i.e. It overwrites all \r or \n or \r\n with 0)!!!)
*/
int bgStringListLines(bgStringList_typ *p);

/**
Method for data object \link bgStringListEx_typ \endlink\n
\param Ptr to data object: (\link bgStringList_typ \endlink)
\param pAddrListBuffer Ptr to memory that will hold list of items (string ptr-s)
\param sizeListBuffer Size of memory (bytes) for list the list of items
*/
void bgStringListExMemSet(bgStringListEx_typ *p, char* pAddrListBuffer, int sizeListBuffer);

/**
Method for data object \link bgStringListEx_typ \endlink\n
\param p Ptr to data object: (\link bgStringListEx_typ \endlink)
\param pContentBuffer Ptr to the input/source stream
\param pAddrListBuffer Ptr to memory that will hold list of items (string ptr-s) (NOTE: if 0, \n
method \link bgStringListExMemSet \endlink must be used prior to calling this method!)
\param sizeListBuffer Size of memory (bytes) for the list of items (NOTE: if 0, \n
method \link bgStringListExMemSet \endlink must be used prior to calling this method!)

<b>IMPORTANT: </b>Method write 0-s (string termination) into the source stream (*pContentBuffer) at the
position of each line end!

See also: \link bgStringListLines \endlink and \link bgStringListExMemSet \endlink
*/
int bgStringListLinesEx(bgStringListEx_typ *p, char* pContentBuffer, char* pAddrListBuffer, int sizeListBuffer);

/**
Method for data object \link bgStringList_typ \endlink\n
\param Ptr to data object: (\link bgStringList_typ \endlink)
Example: Given the input string (*src), i.e.:
\code
"hello world what is new?"
\endcode
Method generates following: (p-> points to \link bgStringList_typ \endlink data object):
\code
p->itemCount = 5; <*src> string has 5 words
p->items[0] = ptr to 1st word ("hello");
p->items[1] = ptr to 2nd word ("world");
p->items[2] = ptr to 3rd word ("what");
p->items[3] = ptr to 4th word ("is");
p->items[4] = ptr to 5th word ("new?");
\endcode
\n
Method is used when processing ascii based client/server protocols (i.e. FTP, Telnet...)\n
<b>IMPORTANT:</b>Method write 0-s (string termination) into the source string (*src) at the position of
each separator!\n
(i.e. It overwrites all seprator characters with 0)!)
*/
int bgStringSplitLine(bgStringList_typ *p, char separator);

/**
Method for data object \link bgStringListEx_typ \endlink\n
\param p Ptr to data object: (\link bgStringListEx_typ \endlink)
\param separator Seperator character (i.e. word separation)
\param pLineBuffer Ptr to the input/source string (stream )
\param pAddrListBuffer Ptr to memory that will hold list of items (string ptr-s) (NOTE: if 0, \n
method \link bgStringListExMemSet \endlink must be used prior to calling this method!)
\param sizeListBuffer Size of memory (bytes) for the list of items (NOTE: if 0, \n
method \link bgStringListExMemSet \endlink must be used prior to calling this method!)

<b>IMPORTANT: </b>Method write 0-s (string termination) into the source string (*pLineBuffer) at the
position of each (separator) character!

See also: \link bgStringSplitLine \endlink and \link bgStringListExMemSet \endlink
*/
int bgStringSplitLineEx(bgStringListEx_typ *p, char separator, char* pLineBuffer, char* pAddrListBuffer, int sizeListBuffer);

/**
Convert string to lower case.
Example: 'Hello'->'hello', 'How Are YOU?'->'how are you?'
\param s Input string
\return Pointer to the same, input string
<b>IMPORTANT: </b>Method modifies the input string (*s) by changing all upper case letters to lower case
letters (if any)!\n
*/
char *bgStringLower(char *s);

/**
Convert string to upper case.
Example: 'Hello'->'HELLO', 'How Are YOU?'->'HOW ARE YOU?'
\param s Input string
\return Pointer to the same, input string
<b>IMPORTANT: </b>Method modifies the input string (*s) by changing all lower case letters to upper case
letters (if any)!\n
*/
char *bgStringUpper(char *s);

/**
Convert character to lower case.
Example: 'H' -> 'h'
\param c Input character
\return Lower case of the input character if possible. If not, returns the same char.
*/
char bgCharToLowerCase(char c);

/**
Compare strings using strcmp.
\param s1 String 1
\param s2 String 2
\param minChrCount not used
\return 0 - if s1 != s2
\return 1 - if s1 == s2
*/
int bgStringIsMatch(char *s1, char *s2, int minChrCount);

/**
Copy part of the source string (*src) to destination (*dest).
\param src Source string ptr
\param StartPosition Defines position in (*src) where the copy begins (src[startPosition])
\param srcEndPosition Defines position in (*src) where the copy ends (src[endPosition - 1])
\param dest Destination buffer
\return Number of bytes copied (i.e. length of the dest string)
NOTE: srcEndPosition is not included in the copy (last copied byte position is srcEndPosition-1)\n
Length of the copied string is (srcEndPosition - srcStartPosition)\n
Example:
\code
src="01234567890"
srcStartPosition=3
srcEndPosition=7
dest="3456"
\endcode
*/
int bgStrCopyFromTo(char* src, int srcStartPosition, int srcEndPosition, char* dest);

/**
Copy source string (*src) to destination (*dest), remove leading/trailing spaces, convert (*dest) to lower
\param src Source string ptr
\param dest Destination buffer
\param maxNoOfCharsToCopy Destination buffer size
\return Number of bytes copied (i.e. length of the dest string)
Example:
\code
src="  0123AB  cdeFG  "
dest="0123ab  cdefg"
\endcode
*/
int bgStrCpyNTrimSpcsToLwr(char *dest, char *src, int maxNoOfCharsToCopy);

/**
Search supplied c string (*src) (zero terminated!!!) for the eol (LF or CRLF).
\param src Source string
\param startPosition Start of the search position
\return Position (>=0) of the EOL character or -1 if EOL not found

*/
int bgStrFindEOL(char* src, int startPosition);

#endif
```

### bgsscanf.c
```c
#ifndef _BG_SSCANF_C
#define _BG_SSCANF_C
/*
Source:
http://www.koders.com/c/fid1D51E1E6F4F922088DF508FFEEEEC702AFED6333.aspx?s=__v_scanf
*/

#define GBLONG_MAX 2147483647L
#define GBLONG_MIN (-GBLONG_MAX-1)
#define GBULONG_MAX (GBLONG_MAX * 2UL + 1)

extern long int strtol ( const char * str, char ** endptr, int base );

#define WANT_FLOATING_POINT_IN_SCANF 1
#define WANT_CHARACTER_CLASSES_IN_SCANF 1

#define	EOF	(-1)

struct arg_scanf {
  void *data;
  int (*getch)(void*);
  int (*putch)(int,void*);
};

struct str_data {
  unsigned char* str;
};

static int sgetc(struct str_data* sd) {
  register unsigned int ret = *(sd->str++);
  return (ret)?(int)ret:-1;
}

static int sputc(int c, struct str_data* sd) {
  return (*(--sd->str)==c)?c:-1;
}

#define A_GETC(fn)	(++consumed,(fn)->getch((fn)->data))
#define A_PUTC(c,fn)	(--consumed,(fn)->putch((c),(fn)->data))

static int isspace(int c)
{
	return ((c==(int)' ')) ? 1 : 0;
}

static int isdigit(int c)
{
	return ((c>=(int)'0') && (c<=(int)'9')) ? 1 : 0;
}

int bg_v_scanf(struct arg_scanf* fn, const unsigned char *format, va_list arg_ptr)
{
  unsigned int ch;	/* format act. char */
  int n=0;

  /* arg_ptr tmps */
#ifdef WANT_FLOATING_POINT_IN_SCANF
  double *pd;
  float  *pf;
#endif
  long   *pl;
  short  *ph;
  int    *pi;
  char    *s;

  unsigned int consumed=0;

  /* get one char */
  int tpch= A_GETC(fn);

  while (*format)
  {
    ch=*format++;
    switch (ch) {
    /* end of format string ?!? */
    case 0: return 0;

    /* skip spaces ... */
    case ' ':
    case '\f':
    case '\t':
    case '\v':
    case '\n':
    case '\r':
      while((*format)&&(isspace(*format))) ++format;
      while(isspace(tpch)) tpch=A_GETC(fn);
      break;

    /* format string ... */
    case '%':
      {
	unsigned int _div=0;
	int width=-1;
	char flag_width=0;
	char flag_discard=0;
	char flag_half=0;
	char flag_long=0;
	char flag_longlong=0;

in_scan:
	ch=*format++;
	if(ch!='n' && tpch==-1) goto err_out;
	switch (ch) {
	/* end of format string ?!? */
	case 0: return 0;

	/* check for % */
	case '%':
	  if ((unsigned char)tpch != ch) goto err_out;
	  tpch=A_GETC(fn);
	  break;

	/* FLAGS */
	case '*':
	  flag_discard=1;
	  goto in_scan;
	case 'h':
	  flag_half=1;
	  goto in_scan;
	case 'l':
	  if (flag_long) flag_longlong=1;
	  flag_long=1;
	  goto in_scan;
	case 'q':
	case 'L':
	  flag_longlong=1;
	  goto in_scan;

	/* WIDTH */
	case '0':
	case '1':
	case '2':
	case '3':
	case '4':
	case '5':
	case '6':
	case '7':
	case '8':
	case '9':
	  width=strtol((const char*)(format-1),&s,10);
	  format=(unsigned char*)s;
	  flag_width=1;
	  goto in_scan;

	/* scan for integer / strtol reimplementation ... */
	case 'p':
	case 'X':
	case 'x':
	  _div+=6;
	case 'd':
	  _div+=2;
	case 'o':
	  _div+=8;
	case 'u':
	case 'i':
	  {
	    unsigned long v=0;
	    unsigned int consumedsofar;
	    int neg=0;
	    while(isspace(tpch)) tpch=A_GETC(fn);
	    if (tpch=='-') {
	      tpch=A_GETC(fn);
	      neg=1;
	    }

	    if (tpch=='+') tpch=A_GETC(fn);

	    if (tpch==-1) return n;
	    consumedsofar=consumed;

	    if (!flag_width) {
	      if ((_div==16) && (tpch=='0')) goto scan_hex;
	      if (!_div) {
		_div=10;
		if (tpch=='0') {
		  _div=8;
scan_hex:
		  tpch=A_GETC(fn);
		  if ((tpch|32)=='x') {
		    tpch=A_GETC(fn);
		    _div=16;
		  }
		}
	      }
	    }
	    while ((width)&&(tpch!=-1)) {
	      register unsigned long c=tpch&0xff;
	      register unsigned long d=c|0x20;
	      c=(d>='a'?d-'a'+10:c<='9'?c-'0':0xff);
	      if (c>=_div) break;
	      d=v*_div;
	      v=(d<v)?GBULONG_MAX:d+c;
	      --width;
	      tpch=A_GETC(fn);
	    }

	    if (consumedsofar==consumed) return n;

	    if ((ch|0x20)<'p') {
	      register long l=v;
	      if (v>=-((unsigned long)GBLONG_MIN)) {
		l=(neg)?GBLONG_MIN:GBLONG_MAX;
	      }
	      else {
		if (neg) v*=-1;
	      }
	    }
	    if (!flag_discard) {
	      if (flag_long) {
		pl=(long *)va_arg(arg_ptr,long*);
		*pl=v;
	      } else if (flag_half) {
		ph=(short*)va_arg(arg_ptr,short*);
		*ph=v;
	      } else {
		pi=(int *)va_arg(arg_ptr,int*);
		*pi=v;
	      }
	      if(consumedsofar<consumed) ++n;
	    }
	  }
	  break;

	/* FIXME: return value of *scanf with ONE float maybe -1 instead of 0 */
#ifdef WANT_FLOATING_POINT_IN_SCANF
	/* floating point numbers */
	case 'e':
	case 'E':
	case 'f':
	case 'g':
	  {
	    double d=0.0;
	    int neg=0;
	    unsigned int consumedsofar;

	    while(isspace(tpch)) tpch=A_GETC(fn);

	    if (tpch=='-') {
	      tpch=A_GETC(fn);
	      neg=1;
	    }
	    if (tpch=='+') tpch=A_GETC(fn);

	    consumedsofar=consumed;

	    while (isdigit(tpch)) {
	      d=d*10+(tpch-'0');
	      tpch=A_GETC(fn);
	    }
	    if (tpch=='.') {
	      double factor=.1;
	      consumedsofar++;
	      tpch=A_GETC(fn);
	      while (isdigit(tpch)) {
		d=d+(factor*(tpch-'0'));
		factor/=10;
		tpch=A_GETC(fn);
	      }
	    }
	    if (consumedsofar==consumed) return n;	/* error */
	    if ((tpch|0x20)=='e') {
	      int exp=0, prec=tpch;
	      double factor=10;
	      tpch=A_GETC(fn);
	      if (tpch=='-') {
		factor=0.1;
		tpch=A_GETC(fn);
	      } else if (tpch=='+') {
		tpch=A_GETC(fn);
	      } else {
		d=0;
		if (tpch!=-1) A_PUTC(tpch,fn);
		tpch=prec;
		goto exp_out;
	      }
	      consumedsofar=consumed;
	      while (isdigit(tpch)) {
		exp=exp*10+(tpch-'0');
		tpch=A_GETC(fn);
	      }
	      if (consumedsofar==consumed) return n;	/* error */
	      while (exp) {	/* as in strtod: XXX: this introduces rounding errors */
		d*=factor; --exp;
	      }
	    }
exp_out:
	    if (!flag_discard) {
	      if (flag_long) {
		pd=(double *)va_arg(arg_ptr,double*);
		*pd=d;
	      } else {
		pf=(float *)va_arg(arg_ptr,float*);
		*pf=d;
	      }
	      ++n;
	    }
	  }
	  break;
#endif

	/* char-sequences */
	case 'c':
	  if (!flag_discard) {
	    s=(char *)va_arg(arg_ptr,char*);
	    ++n;
	  }
	  if (!flag_width) width=1;
	  while (width && (tpch!=-1)) {
	    if (!flag_discard) *(s++)=tpch;
	    --width;
	    tpch=A_GETC(fn);
	  }
	  break;

	/* string */
	case 's':
	  if (!flag_discard) s=(char *)va_arg(arg_ptr,char*);
	  while(isspace(tpch)) tpch=A_GETC(fn);
	  if (tpch==-1) break;		/* end of scan -> error */
	  while (width && (tpch!=-1) && (!isspace(tpch))) {
	    if (!flag_discard) *s=tpch;
	    if (tpch) ++s; else break;
	    --width;
	    tpch=A_GETC(fn);
	  }
	  if (!flag_discard) { *s=0; ++n; }
	  break;

	/* consumed-count */
	case 'n':
	  if (!flag_discard) {
	    pi=(int *)va_arg(arg_ptr,int *);
            *pi=consumed-1;
	  }
	  break;

#ifdef WANT_CHARACTER_CLASSES_IN_SCANF
	case '[':
	  {
	    char cset[256];
	    int flag_not=0;
	    int flag_dash=0;
	    brsmemset((UDINT)cset,0,sizeof(cset));
	    ch=*format++;
	    /* first char specials */
	    if (ch=='^') {
	      flag_not=1;
	      ch=*format++;
	    }
	    if ((ch=='-')||(ch==']')) {
	      cset[ch]=1;
	      ch=*format++;
	    }
	    /* almost all non special chars */
	    for (;(*format) && (*format!=']');++format) {
	      if (flag_dash) {
		register unsigned char tmp=*format;
		for (;ch<=tmp;++ch) cset[ch]=1;
		flag_dash=0;
		ch=*format;
	      }
	      else if (*format=='-') flag_dash=1;
	      else {
		cset[ch]=1;
		ch=*format;
	      }
	    }
	    /* last char specials */
	    if (flag_dash) cset['-']=1;
	    else cset[ch]=1;

	    /* like %c or %s */
	    if (!flag_discard) {
	      s=(char *)va_arg(arg_ptr,char*);
	      ++n;
	    }
	    while (width && (tpch>=0) && (cset[tpch]^flag_not)) {
	      if (!flag_discard) *s=tpch;
	      if (tpch) ++s; else break;
	      --width;
	      tpch=A_GETC(fn);
	    }
	    if (!flag_discard) *s=0;
	    ++format;
	  }
	  break;
#endif
	default:
	  goto err_out;
	}
      }
      break;

    /* check if equal format string... */
    default:
      if ((unsigned char)tpch != ch) goto err_out;
      tpch=A_GETC(fn);
      break;
    }
  }

  /* maybe a "%n" follows */
  if(*format) {
    while(isspace(*format)) format++;
    if(format[0] == '%' && format[1] == 'n') {
      pi = (int *) va_arg(arg_ptr, int *);
      *pi = consumed - 1;
    }
  }

err_out:
  if (tpch<0 && n==0) return EOF;
  A_PUTC(tpch,fn);
  return n;
}

int bgvsscanf(const char* str, const  char* format, va_list arg_ptr)
{
  struct str_data  fdat = { (unsigned char*)str };
  struct arg_scanf farg = { (void*)&fdat, (int(*)(void*))sgetc, (int(*)(int,void*))sputc };
  return bg_v_scanf(&farg, (unsigned char*) format, arg_ptr);
}

int bgsscanf(const char *str, const char *format, ...)
{
  int n;
  va_list arg_ptr;
  va_start(arg_ptr, format);
  n=bgvsscanf(str,format,arg_ptr);
  va_end (arg_ptr);
  return n;
}

#endif
```

### Package Logical/paiComponents/paiFileService - pai File Access service package

### paiFSInterface.h
```c
/********************************************************************
 * COPYRIGHT --
 ********************************************************************
 * Package: paiFileService
 * File: paFSInterface.h
 * Author: goran
 * Created: August 18, 2015
 *******************************************************************/

#include <bur/plctypes.h>

BOOL paiFSFileRequestIsBusy(paiFileService_typ* p);
BOOL paiFSFileSystemIsInit(paiFileService_typ* p);
void paiFSExeCallback(paiFileService_typ* p);
void paiFSExeCallbackCyclic(paiFileService_typ* p);
void paiFSSetCallback(paiFileService_typ* p, UDINT pCallback, UDINT pCallbackData);
void paiFSDirCreateRequest(paiFileService_typ* p, UDINT adrDeviceName, UDINT adrDirPath, UDINT pCallback, UDINT pCallbackData);
void paiFSDirInfoRequest(paiFileService_typ* p, UDINT adrDeviceName, UDINT adrDirPath, UDINT pCallback, UDINT pCallbackData);
void paiFSFileDelRequest(paiFileService_typ* p, UDINT adrDeviceName, UDINT adrFilePath, UDINT pCallback, UDINT pCallbackData);
void paiFSFileRdRequest(paiFileService_typ* p, UDINT adrDeviceName, UDINT adrFilePath, UDINT adrDst, UDINT sizeDst, UDINT pCallback, UDINT pCallbackData);
void paiFSFileWrRequest(paiFileService_typ* p, UDINT adrDeviceName, UDINT adrFilePath, UDINT adrSrc, UDINT sizeSrc, UDINT pCallback, UDINT pCallbackData);
//EOF
```

### Package Logical/paiComponents/paiHmi - pai HMI related components

### paiHmiMsgScroll.typ
```iecst
(********************************************************************
 * COPYRIGHT -- pai
 ********************************************************************
 * Package: HMI
 * File: HMI.typ
 * Author: goran
 * Created: August 28, 2013
 ********************************************************************
 * Data types of package HMI
 ********************************************************************)
(*########################################################################*)
(*HMI object - Scrolling Messages (i.e. alarms)*)
(*########################################################################*)

TYPE
	paiHmiMsgScrolling_typ : 	STRUCT  (*0-disable; 1-enable*)
		iEnable : BOOL; (*input: address of the alarm array*)
		iAdrAlarmArray : UDINT; (*input: address of the alarm array*)
		iAlarmArrayLen : UDINT; (*input: number of alarms in the alarm array*)
		iMsgTimeXms : UDINT; (*input: duration of the message display (if more than one message/alarm active)*)
		oMsgID : UINT; (*output: message ID of the active alarm / message*)
		oMsgVisible : UINT; (*output: visibilty control DP for the VC text message*)
		state : UINT; (*Status for common dialog layer*)
		tmr1 : TON; (*Dialog control timer*)
	END_STRUCT;
END_TYPE
```

### paiHmiTemplate.typ
```iecst
(********************************************************************
 * COPYRIGHT --
 ********************************************************************
 * Package: HMI
 * File: cfgPaiHmiTemplate.typ
 * Author: goran
 * Created: October 15, 2014
 ********************************************************************
 * Data types of package HMI
 ********************************************************************)
(*########################################################################*)
(*HMI key assinged PV-s (i.e. page navigation, save btns, etc)*)
(*########################################################################*)

TYPE
	paiHmiTemplateEnums_typ :
		(
		paiHMI_ENUM_MENU_ITEMS_LT := 10, (*Main menu - left side - number of buttons*)
		paiHMI_ENUM_TABS_MAXIDX := 10, (*Max number of tab keys per page*)
		paiHMI_ENUM_TG_TEXT_MAXIDX := 127, (*Max number of lines in the Text Group for Page Navigation*)
		paiHMI_ENUM_TG_TEXT_MAXLEN := 31, (*Max number of lines in the Text Group for Page Navigation*)
		paiHMI_PWD_LEVELS := 5, (*Number of password levels (0-operator;1-supervisor;2-admin;3-maintenance;4-factory)*)
		paiHMI_PWD_MAXLEN := 15 (*Max pwd len*)
		);
END_TYPE

(*########################################################################*)
(*HMI key assinged PV-s (i.e. menu, tabs, etc)*)
(*########################################################################*)

TYPE
	paiHmiTemplateKeys_typ : 	STRUCT
		menuKeyTopLT : INT; (*Menu key press top LF*)
		menuKeyTopRT : INT; (*Mom keys connected to menu items RT*)
		currentMenuLF : INT;
		currentMenuRT : INT;
		tabKeysRadioDataPoint : INT; (*DP that tab button are writing to in order to create radio buttons/tab view effect*)
		tabKeysRadioDataPointOld : INT; (*DP that tab button are writing to in order to create radio buttons/tab view effect*)
		tabKeysRadioArray : ARRAY[0..paiHMI_ENUM_TABS_MAXIDX]OF INT;
	END_STRUCT;
END_TYPE

(*########################################################################*)
(*HMI related status control PV-s (i.e. visibility, locking, etc)*)
(*########################################################################*)

TYPE
	paiHmiTemplateStatus_typ : 	STRUCT
		menuVisibleLT : UINT; (*Main menu LF visibility control *)
		menuIndexLT : UINT; (*Main menu currently selected menu item - LF*)
		loginVisibleGE1 : USINT; (*Visibility control for login level related stuff - set to visible (0) if login level >= 1; othervise set to 1 (i.e. loginLevel < 1)*)
		loginVisibleGE2 : USINT; (*Visibility control for login level related stuff - set to visible (0) if login level >= 2; othervise set to 1 (i.e. loginLevel < 2)*)
		menuLFHideTimer : TON; (*timer of automaticaly hiding LF dropdown menu*)
		unusedItemInvisible : UDINT; (*used for VC items that are not used (hidden)*)
		passwordStrings : ARRAY[0..paiHMI_PWD_LEVELS]OF STRING[paiHMI_PWD_MAXLEN]; (*Password strings used for loginLevel control*)
	END_STRUCT;
END_TYPE

(*########################################################################*)
(*HMI related timer settings*)
(*########################################################################*)

TYPE
	paiHmiTemplateTimerSettings_typ : 	STRUCT
		loginTimeout : REAL; (*Login timeout timer setting*)
		dialogBoxTimeout : REAL; (*Dialog box (i.e. save data? yes/no) timeout for waiting on input*)
		splashScreenTimeout : REAL; (*Duration of the initial screen (i.e. manufacturer logo) *)
		dropdwMenuLFTimeout : REAL; (*Duration after which a dropdown menu is automaticaly hiden if not clicked *)
	END_STRUCT;
END_TYPE

(*########################################################################*)
(*HMI pwd settings*)
(*########################################################################*)

TYPE
	paiHmiTemplatePwdSettings_typ : 	STRUCT
		passwordAdmin : STRING[paiHMI_PWD_MAXLEN]; (*Login timeout timer setting*)
		passwordMaint : STRING[paiHMI_PWD_MAXLEN]; (*Login timeout timer setting*)
		passwordSupervisor : STRING[paiHMI_PWD_MAXLEN]; (*Login timeout timer setting*)
		passwordFactory : STRING[paiHMI_PWD_MAXLEN]; (*Login timeout timer setting*)
	END_STRUCT;
END_TYPE

(*########################################################################*)
(*HMI related PV-s connected to VC runtime (see VC runtime settings)*)
(*########################################################################*)

TYPE
	paiHmiTemplateVCRuntime_typ : 	STRUCT
		wheelCount : INT;
		wheelEnter : INT;
		keyLevelChange : INT;
		keyLevelCurrent : INT;
		languageChange : INT;
		languageCurrent : INT;
		keyMatrix : ARRAY[0..63]OF INT;
		LEDMatrix : ARRAY[0..63]OF INT;
		pageChange : INT;
		pageCurrent : INT;
		lifeSign : INT;
		IPAddress : STRING[31];
		focusControl : INT;
		helpControl : INT;
		touchCalibration : INT;
		touchCalibrationState : INT;
		screenSaverTimeout_sec : INT;
		screenSaverPage : INT;
	END_STRUCT;
END_TYPE

(*########################################################################*)
(*HMI related config file settings*)
(*########################################################################*)

TYPE
	paiHmiTemplateConfig_typ : 	STRUCT
		pwdSettings : paiHmiTemplatePwdSettings_typ;
		timerSettings : paiHmiTemplateTimerSettings_typ;
	END_STRUCT;
END_TYPE

(*########################################################################*)
(*HMI control logic private PV-s*)
(*########################################################################*)

TYPE
	paiHmiTemplateItem_typ : 	STRUCT
		itemText : STRING[31];
		itemVisible : UINT;
		itemDisabled : UINT;
		jumpPageId : UINT;
	END_STRUCT;
	paiHmiTemplateSubmenuItem_typ : 	STRUCT
		button : paiHmiTemplateItem_typ;
		tabs : ARRAY[0..paiHMI_ENUM_TABS_MAXIDX]OF paiHmiTemplateItem_typ;
	END_STRUCT;
	paiHmiTemplatePrivate_typ : 	STRUCT
		initDone : BOOL;
		state : INT;
		vcHandle : UDINT;
		index : UDINT;
		indexButton : UDINT;
		indexTab : UDINT;
		TG_id : UDINT;
		text : STRING[paiHMI_ENUM_TG_TEXT_MAXLEN];
		parseErrorText : STRING[127];
		textLen : UINT;
		textLines : ARRAY[0..paiHMI_ENUM_TG_TEXT_MAXIDX]OF STRING[paiHMI_ENUM_TG_TEXT_MAXLEN];
		activeTabs : ARRAY[0..paiHMI_ENUM_TABS_MAXIDX]OF paiHmiTemplateItem_typ;
		menuLF : ARRAY[0..paiHMI_ENUM_MENU_ITEMS_LT]OF paiHmiTemplateSubmenuItem_typ;
		pageSetByLFMenu : INT;
		pageCurrent : UDINT;
		pagePrev : UDINT;
		pageInit : BOOL;
		pageExit : BOOL;
	END_STRUCT;
	paiHmiTemplate_typ : 	STRUCT
		runtime : paiHmiTemplateVCRuntime_typ; (*VC runtime Datapoint PV-s. Assigned to different VC control points.*)
		status : paiHmiTemplateStatus_typ;
		keys : paiHmiTemplateKeys_typ;
		timerSettings : paiHmiTemplateTimerSettings_typ;
		activeTabs : ARRAY[0..paiHMI_ENUM_TABS_MAXIDX]OF paiHmiTemplateItem_typ;
		activeTopMenuLF : paiHmiTemplateItem_typ;
		currentMenuLF : INT;
		currentTab : INT;
		prv : paiHmiTemplatePrivate_typ;
	END_STRUCT;
END_TYPE
```


- Program Logical/paiComponents/paiTelnet/paiTelnet (ANSIC) (no source held here)

### Package Logical/paiComponents/paiTemplate - pai Template Application with Drop down menues and tabs page navigation

### paiHMI.var
```iecst
(********************************************************************
 * COPYRIGHT -- pai
 ********************************************************************
 * Package: HMI
 * File: HMI.var
 * Author: goran
 * Created: August 28, 2013
 ********************************************************************
 * Variables of package HMI
 ********************************************************************)
VAR
	gHmiParamTable : hmiParamListTable_typ; (*Machine configuration / parameter settings logic *)
	gPaiHmiMain : paiHmiTemplate_typ; (*HMI logic, page navigation, visibility control, etc.*)
	gPaiHmiMsgScroll : paiHmiMsgScrolling_typ; (*Scrolling Alarm Msg Support*)
	gPaiHmiDialogMsg : paiHmiDialog_typ; (*Scrolling Alarm Msg Support*)
	gPaiHmiAlertMsg : paiHmiAlert_typ; (*Scrolling Alarm Msg Support*)
	gPaiHmiRTMenu : paiHmiDropdwMenuRT_typ;
	gPaiHmiSystemDateTime : paiHmiSystemTime_typ;
	gPaiHmiNetworking : paiHmiSystemNetworking_typ;
END_VAR
VAR RETAIN
	gScrensaverTimeout : INT := 0;
END_VAR
```

- MpPMLStateColors.clm (not shown)

- stationStatus.clm (not shown)

- Arial12px.fninfo (not shown)

- Arial9px.fninfo (not shown)

- Button.fninfo (not shown)

- Header.fninfo (not shown)

- Input.fninfo (not shown)

- MenuItemsSmall.fninfo (not shown)

- Status.fninfo (not shown)

- dialogMsg.layer (not shown)

- paiHmiMenu.layer (not shown)

- paiMpRecipeMsgBox.layer (not shown)

- AlphaPad.tpr (not shown)

- AlphaPad2.tpr (not shown)

- NumPad.tpr (not shown)

### Package Logical/paiComponents/paiUtility - pai defined types 

### paiBnRVFD.typ
```iecst
(********************************************************************

 * COPYRIGHT -- Piedmont Automation Inc.

 ********************************************************************

 * File: MachineIO.typ

 * Author: goran

 * Created: Jun 1, 2015

 ********************************************************************

 *)
(*********************************************************************************

B&R VFD related IO Structures
In - direction from VFD to PLC
Out - direction from PLC to VFD

*********************************************************************************)
(**)

TYPE
	paiVFDInFault_typ : 	STRUCT
		FaultCounter : UINT;
		CurrentFault : UINT; (*CiA402 fault code*)
		CurrentFaultTxt : STRING[63];
		LastFault : INT; (*Last dedected fault*)
	END_STRUCT;
	paiVFDInIO_typ : 	STRUCT  (*Logic inputs states*)
		LogicInput1 : BOOL; (*Logic inputs states (Value of LI1)*)
		LogicInput2 : BOOL; (*Logic inputs states (Value of LI2)*)
		LogicInput3 : BOOL; (*Logic inputs states (Value of LI3)*)
		LogicInput4 : BOOL; (*Logic inputs states (Value of LI4)*)
		LogicInput5 : BOOL;
		LogicInput6 : BOOL;
		Relay01State : BOOL;
		Relay02State : BOOL;
		AnalogInput1 : INT;
		AnalogInput2 : INT;
	END_STRUCT;
	paiVFDInStatus_typ : 	STRUCT  (*Status words*)
		SpeedMode : BOOL;
		PowerRemoval : BOOL;
		ReadyToSwitchOn : BOOL; (*(1 = Ready to switch on)*)
		SwitchedOn : BOOL; (*(1 = Switched on, ready)*)
		OperationEnabled : BOOL; (*(1 = Operation enabled, running)*)
		FaultDetection : BOOL; (*(1 = Fault detection)*)
		VoltageEnabled : BOOL; (*(Voltage disabled, always = 0)*)
		QuickStop : BOOL; (*(0 = Quick stop, emergency stop)*)
		SwitchOnDisabled : BOOL; (*(1 = Switched on disabled)	*)
		WarningAlarm : BOOL; (*(1 = Alarm)*)
		TargetReached : BOOL; (*(1 = Target reached, reference reached)*)
		StopKey : BOOL; (*(1 = Stop via STOP key)*)
		Direction : BOOL; (*(Direction of rotation 0 = Forward rotation; 1 = Reverse rotation)*)
		Accelerating : BOOL; (*(1 = Acceleration in progress)*)
		Decelerating : BOOL; (*(1 = Deceleration in progress)*)
		FastStop : BOOL; (*(1 = Fast stop in progress)*)
		CurrentVelocity : INT; (*Output velocity [rpm]*)
		MotorTorque : INT; (*Motor torque [%]*)
		MotorCurrent : UINT; (*Motor current [0.1 A]*)
		DriveThermalState : UINT; (*Drive thermal state [%]*)
		MotorThermalState : UINT; (*Motor thermal state [%]*)
	END_STRUCT;
	paiVFDIn_typ : 	STRUCT
		ModuleInfo : paiBnRHWModuleInfo_typ;
		IO : paiVFDInIO_typ;
		Status : paiVFDInStatus_typ;
		Fault : paiVFDInFault_typ;
	END_STRUCT;
	paiVFDOutControl_typ : 	STRUCT  (*Control words*)
		SwitchOn : BOOL; (* (1 = Switch on)*)
		DisableVoltage : BOOL; (*(0 = Disable voltage)*)
		QuickStop : BOOL; (*(0 = Quick stop/Emergency stop)*)
		EnableOperation : BOOL; (*(1 = Enable operation/Run command)*)
		FaultReset : BOOL; (*(Fault reset/Fault acknowledgment active on 0 V 1 rising edge)*)
		RunAsked : BOOL;
		Direction : BOOL; (*(0 = Forward rotation; 1 = Reverse rotation)*)
		FastStop : BOOL; (*Stop command (0 = No action; 1 = Depending on the STT Type of stop parameter)*)
		DCInjectionBraking : BOOL;
		VelocitySetpoint : INT; (*Speed setpoint [rpm]*)
		TorqueSetpoint : INT;
		TorqueMode : BOOL;
	END_STRUCT;
	paiVFDOutIO_typ : 	STRUCT
		Relay1 : BOOL;
		Relay2 : BOOL;
		AnalogOut1 : INT;
		LogicOut1 : BOOL;
	END_STRUCT;
	paiVFDOut_typ : 	STRUCT
		Control : paiVFDOutControl_typ;
		IO : paiVFDOutIO_typ;
	END_STRUCT;
	paiVFDApplicationIF_typ : 	STRUCT
		iVoltageEnable : BOOL;
		iEnable : BOOL;
		iMoveFwd : BOOL;
		iMoveRev : BOOL;
		iEStop : BOOL;
		iRampStop : BOOL;
		iFaultReset : BOOL;
		iVelocitySetPoint : INT;
		iTorqueSetPoint : INT;
		oReady : BOOL;
		oRunning : BOOL;
		oFault : BOOL;
	END_STRUCT;
	paiVFD_typ : 	STRUCT
		description : STRING[79];
		location : STRING[79];
		stateText : STRING[31];
		appID : UDINT;
		vfdCtrl : paiVFDApplicationIF_typ;
		vfdIn : paiVFDIn_typ;
		vfdOut : paiVFDOut_typ;
	END_STRUCT;
END_TYPE
```

- Program Logical/paiComponents/LibAsUSB1_ST/read_data (IEC) (no source held here)

### X64param.var
```iecst
(********************************************************************
 * COPYRIGHT --
 ********************************************************************
 * Program: X64param
 * File: X64param.var
 * Author: scoccimaroj
 * Created: July 14, 2010
 ********************************************************************
 * Local variables of program X64param
 ********************************************************************)
VAR
	cmdStart : BOOL; (*Start command*)
	State : USINT; (*state machine state*)
	i : UINT; (*counter variable*)
	AsIOAccRead_0 : AsIOAccRead; (*Read function block*)
	csvSearch : CSV_Search;
	csvWrite : CSV_WriteFile;
	csvInit : CSV_Init;
	csvInitCheckFile : CSV_InitCheckFile;
	pNames : ARRAY[0..4] OF UDINT;
	csvStrucMem : UDINT;
	csvMemLength : UDINT;
	position : INT;
END_VAR
```

### Program Logical/Simulation/counter2 (ANSIC) - A new program

#### counter2.c - Implementation code
```c
/********************************************************************
 * COPYRIGHT -- HP
 ********************************************************************
 * Program: counter2
 * File: counter2.c
 * Author: goran
 * Created: March 07, 2013
 ********************************************************************
 * Implementation of program counter2
 ********************************************************************/

#include <bur/plctypes.h>

#ifdef _DEFAULT_INCLUDES
	#include <AsDefault.h>
#endif

_LOCAL int counter2;

void _INIT counter2INIT(void)
{
	/* TODO: Add code here */
}

void _CYCLIC counter2CYCLIC(void)
{
	/* TODO: Add code here */
	counter2++;
}
```

Listed in the project but not available here: Logical/paiComponents/paiMp, Logical/paiComponents/paiTelnet/paiTelnet/paiTelnet.c, Logical/paiComponents/bglib/bgTelnetSrvr-astcpV2.c, Logical/paiComponents/bglib/bgringbuffer.c, Logical/paiComponents/bglib/bgstring.c, Logical/paiComponents/paiPing, Logical/paiComponents/paiUser, Logical/paiComponents/paiUDP, Logical/paiComponents/paiUtility/paiBnRHW.typ, Logical/paiComponents/paiUtility/paiProjectInfo.typ, Logical/paiComponents/LibAsUSB1_ST/read_data/read_data.st, Logical/paiComponents/LibAsUSB1_ST/read_data/read_data.typ, Logical/paiComponents/LibAsUSB1_ST/read_data/read_data.var, Logical/Simulation/Simulation.typ, Logical/Simulation/Simulation.var, Logical/Simulation/simonly, Logical/Simulation/counter, Logical/Simulation/IOsim
